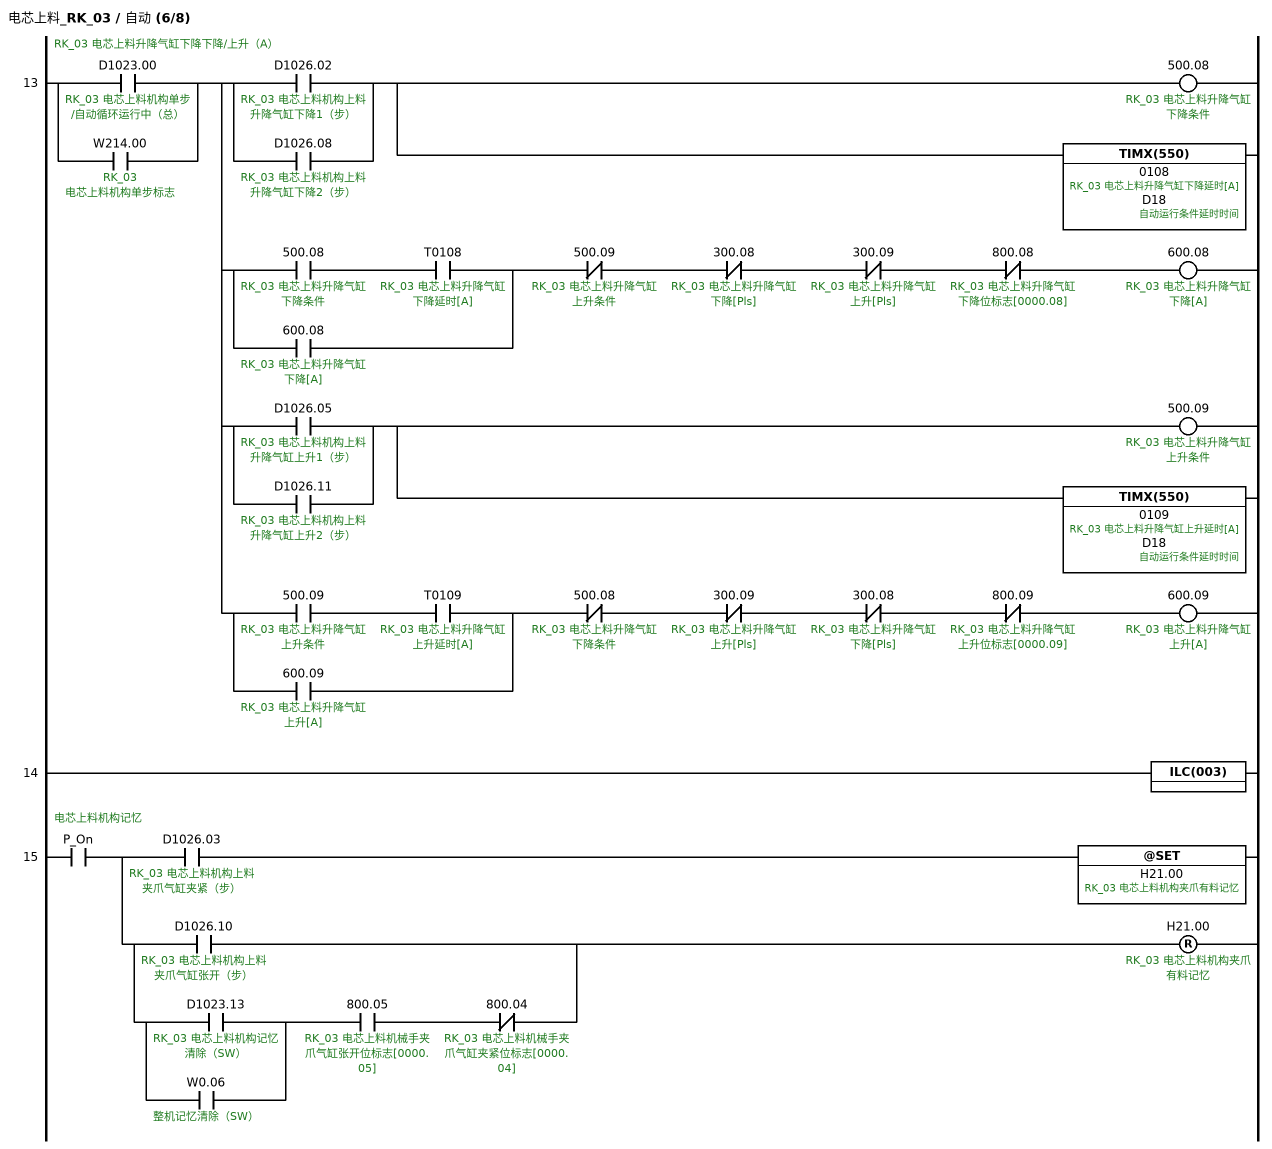
; [picture p384: 电芯上料_RK_03 / 自动, rungs 13-15]
; rung 13: RK_03 电芯上料升降气缸下降下降/上升（A）
LD D1023.00  ; RK_03 电芯上料机构单步/自动循环运行中（总）
OR W214.00  ; RK_03  电芯上料机构单步标志
OUT TR0
LD D1026.02  ; RK_03 电芯上料机构上料升降气缸下降1（步）
OR D1026.08  ; RK_03 电芯上料机构上料升降气缸下降2（步）
ANDLD
OUT 500.08  ; RK_03 电芯上料升降气缸下降条件
TIMX(550) 0108 D18  ; 自动运行条件延时时间, RK_03 电芯上料升降气缸下降延时[A]
LD TR0
LD 500.08  ; RK_03 电芯上料升降气缸下降条件
AND T0108  ; RK_03 电芯上料升降气缸下降延时[A]
OR 600.08  ; RK_03 电芯上料升降气缸下降[A]
ANDLD
ANDNOT 500.09  ; RK_03 电芯上料升降气缸上升条件
ANDNOT 300.08  ; RK_03 电芯上料升降气缸下降[Pls]
ANDNOT 300.09  ; RK_03 电芯上料升降气缸上升[Pls]
ANDNOT 800.08  ; RK_03 电芯上料升降气缸下降位标志[0000.08]
OUT 600.08  ; RK_03 电芯上料升降气缸下降[A]
LD TR0
LD D1026.05  ; RK_03 电芯上料机构上料升降气缸上升1（步）
OR D1026.11  ; RK_03 电芯上料机构上料升降气缸上升2（步）
ANDLD
OUT 500.09  ; RK_03 电芯上料升降气缸上升条件
TIMX(550) 0109 D18  ; 自动运行条件延时时间, RK_03 电芯上料升降气缸上升延时[A]
LD TR0
LD 500.09  ; RK_03 电芯上料升降气缸上升条件
AND T0109  ; RK_03 电芯上料升降气缸上升延时[A]
OR 600.09  ; RK_03 电芯上料升降气缸上升[A]
ANDLD
ANDNOT 500.08  ; RK_03 电芯上料升降气缸下降条件
ANDNOT 300.09  ; RK_03 电芯上料升降气缸上升[Pls]
ANDNOT 300.08  ; RK_03 电芯上料升降气缸下降[Pls]
ANDNOT 800.09  ; RK_03 电芯上料升降气缸上升位标志[0000.09]
OUT 600.09  ; RK_03 电芯上料升降气缸上升[A]
; rung 14
ILC(003)
; rung 15: 电芯上料机构记忆
LD P_On
OUT TR0
AND D1026.03  ; RK_03 电芯上料机构上料夹爪气缸夹紧（步）
@SET H21.00  ; RK_03 电芯上料机构夹爪有料记忆
LD TR0
LD D1026.10  ; RK_03 电芯上料机构上料夹爪气缸张开（步）
LD D1023.13  ; RK_03 电芯上料机构记忆清除（SW）
OR W0.06  ; 整机记忆清除（SW）
AND 800.05  ; RK_03 电芯上料机械手夹爪气缸张开位标志[0000.05]
ANDNOT 800.04  ; RK_03 电芯上料机械手夹爪气缸夹紧位标志[0000.04]
ORLD
ANDLD
RSET H21.00  ; RK_03 电芯上料机构夹爪有料记忆

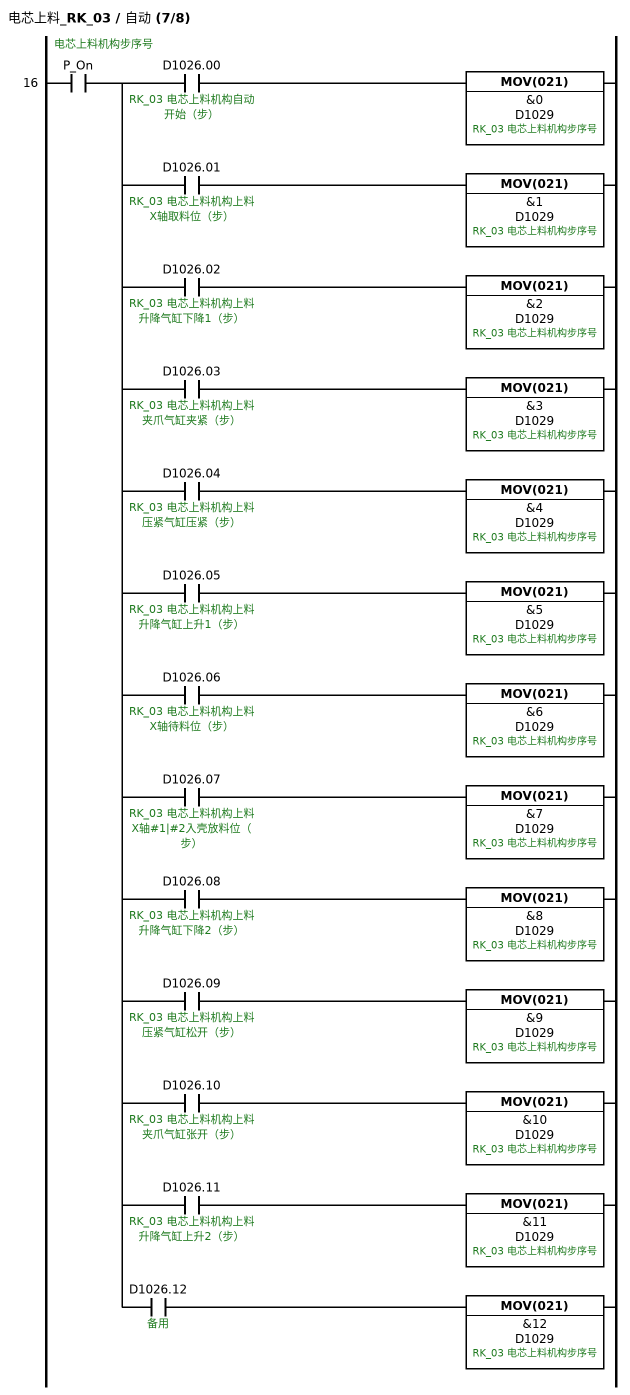
; rung 16: 电芯上料机构步序号
LD P_On
OUT TR0
AND D1026.00  ; RK_03 电芯上料机构自动开始（步）
MOV(021) &0 D1029  ; RK_03 电芯上料机构步序号
LD TR0
AND D1026.01  ; RK_03 电芯上料机构上料X轴取料位（步）
MOV(021) &1 D1029  ; RK_03 电芯上料机构步序号
LD TR0
AND D1026.02  ; RK_03 电芯上料机构上料升降气缸下降1（步）
MOV(021) &2 D1029  ; RK_03 电芯上料机构步序号
LD TR0
AND D1026.03  ; RK_03 电芯上料机构上料夹爪气缸夹紧（步）
MOV(021) &3 D1029  ; RK_03 电芯上料机构步序号
LD TR0
AND D1026.04  ; RK_03 电芯上料机构上料压紧气缸压紧（步）
MOV(021) &4 D1029  ; RK_03 电芯上料机构步序号
LD TR0
AND D1026.05  ; RK_03 电芯上料机构上料升降气缸上升1（步）
MOV(021) &5 D1029  ; RK_03 电芯上料机构步序号
LD TR0
AND D1026.06  ; RK_03 电芯上料机构上料X轴待料位（步）
MOV(021) &6 D1029  ; RK_03 电芯上料机构步序号
LD TR0
AND D1026.07  ; RK_03 电芯上料机构上料X轴#1|#2入壳放料位（步）
MOV(021) &7 D1029  ; RK_03 电芯上料机构步序号
LD TR0
AND D1026.08  ; RK_03 电芯上料机构上料升降气缸下降2（步）
MOV(021) &8 D1029  ; RK_03 电芯上料机构步序号
LD TR0
AND D1026.09  ; RK_03 电芯上料机构上料压紧气缸松开（步）
MOV(021) &9 D1029  ; RK_03 电芯上料机构步序号
LD TR0
AND D1026.10  ; RK_03 电芯上料机构上料夹爪气缸张开（步）
MOV(021) &10 D1029  ; RK_03 电芯上料机构步序号
LD TR0
AND D1026.11  ; RK_03 电芯上料机构上料升降气缸上升2（步）
MOV(021) &11 D1029  ; RK_03 电芯上料机构步序号
LD TR0
AND D1026.12  ; 备用
MOV(021) &12 D1029  ; RK_03 电芯上料机构步序号

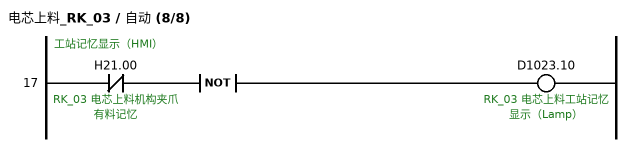
; rung 17: 工站记忆显示（HMI）
LDNOT H21.00  ; RK_03 电芯上料机构夹爪有料记忆
NOT(520)
OUT D1023.10  ; RK_03 电芯上料工站记忆显示（Lamp）

### Section 复位

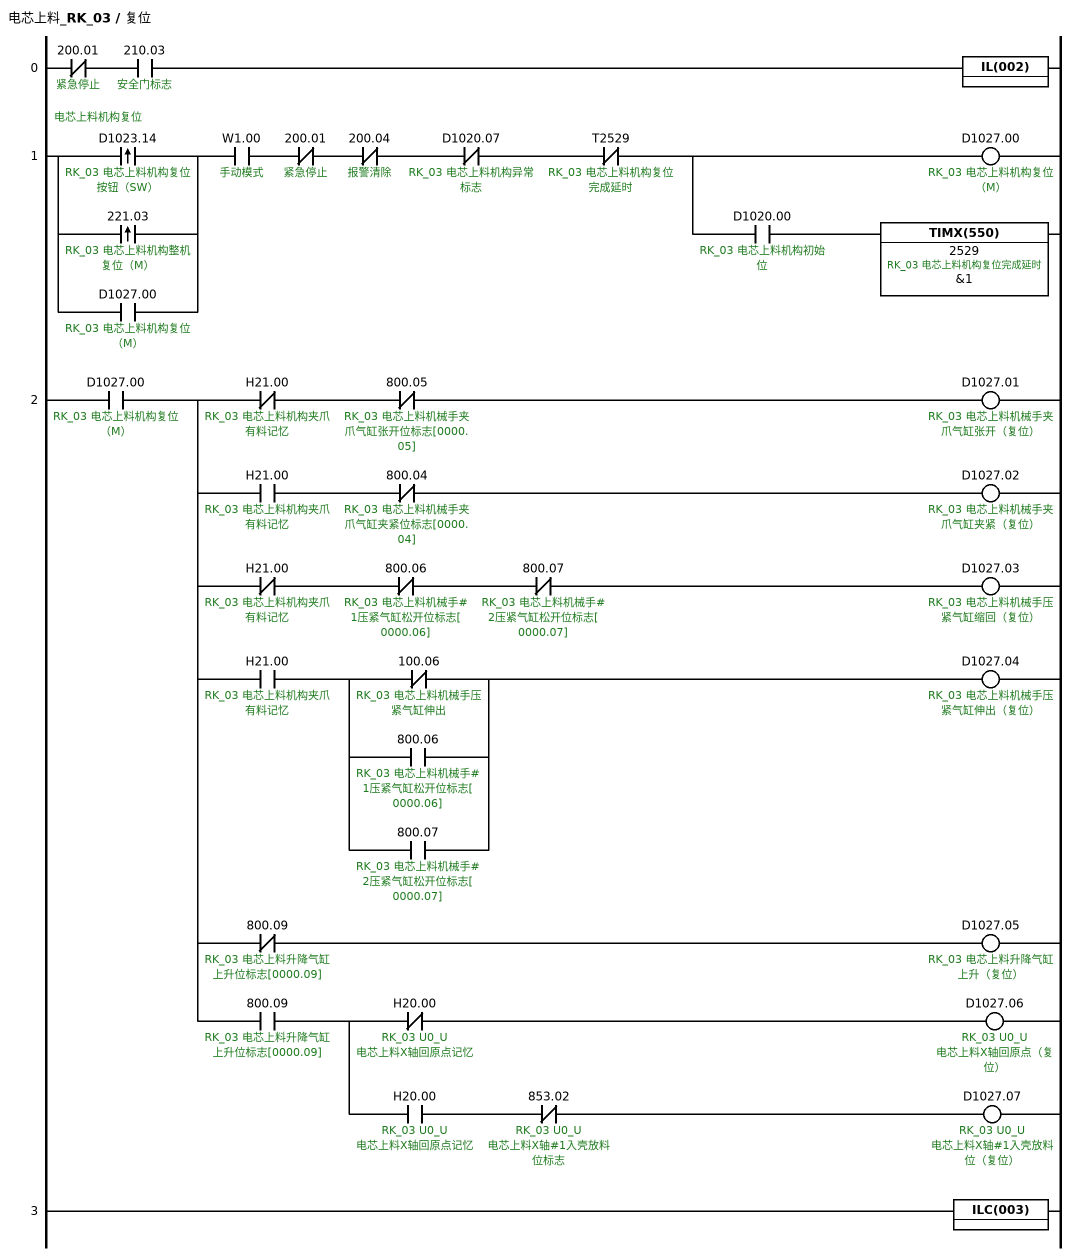
; rung 0
LDNOT 200.01  ; 紧急停止
AND 210.03  ; 安全门标志
IL(002)
; rung 1: 电芯上料机构复位
@LD D1023.14  ; RK_03 电芯上料机构复位按钮（SW）
@OR 221.03  ; RK_03 电芯上料机构整机复位（M）
OR D1027.00  ; RK_03 电芯上料机构复位（M）
AND W1.00  ; 手动模式
ANDNOT 200.01  ; 紧急停止
ANDNOT 200.04  ; 报警清除
ANDNOT D1020.07  ; RK_03 电芯上料机构异常标志
ANDNOT T2529  ; RK_03 电芯上料机构复位完成延时
OUT D1027.00  ; RK_03 电芯上料机构复位（M）
AND D1020.00  ; RK_03 电芯上料机构初始位
TIMX(550) 2529 &1  ; RK_03 电芯上料机构复位完成延时
; rung 2
LD D1027.00  ; RK_03 电芯上料机构复位（M）
OUT TR0
ANDNOT H21.00  ; RK_03 电芯上料机构夹爪有料记忆
ANDNOT 800.05  ; RK_03 电芯上料机械手夹爪气缸张开位标志[0000.05]
OUT D1027.01  ; RK_03 电芯上料机械手夹爪气缸张开（复位）
LD TR0
AND H21.00  ; RK_03 电芯上料机构夹爪有料记忆
ANDNOT 800.04  ; RK_03 电芯上料机械手夹爪气缸夹紧位标志[0000.04]
OUT D1027.02  ; RK_03 电芯上料机械手夹爪气缸夹紧（复位）
LD TR0
ANDNOT H21.00  ; RK_03 电芯上料机构夹爪有料记忆
ANDNOT 800.06  ; RK_03 电芯上料机械手#1压紧气缸松开位标志[0000.06]
ANDNOT 800.07  ; RK_03 电芯上料机械手#2压紧气缸松开位标志[0000.07]
OUT D1027.03  ; RK_03 电芯上料机械手压紧气缸缩回（复位）
LD TR0
AND H21.00  ; RK_03 电芯上料机构夹爪有料记忆
LDNOT 100.06  ; RK_03 电芯上料机械手压紧气缸伸出
OR 800.06  ; RK_03 电芯上料机械手#1压紧气缸松开位标志[0000.06]
OR 800.07  ; RK_03 电芯上料机械手#2压紧气缸松开位标志[0000.07]
ANDLD
OUT D1027.04  ; RK_03 电芯上料机械手压紧气缸伸出（复位）
LD TR0
ANDNOT 800.09  ; RK_03 电芯上料升降气缸上升位标志[0000.09]
OUT D1027.05  ; RK_03 电芯上料升降气缸上升（复位）
LD TR0
AND 800.09  ; RK_03 电芯上料升降气缸上升位标志[0000.09]
OUT TR0
ANDNOT H20.00  ; RK_03 U0_U 电芯上料X轴回原点记忆
OUT D1027.06  ; RK_03 U0_U 电芯上料X轴回原点（复位）
LD TR0
AND H20.00  ; RK_03 U0_U 电芯上料X轴回原点记忆
ANDNOT 853.02  ; RK_03 U0_U 电芯上料X轴#1入壳放料位标志
OUT D1027.07  ; RK_03 U0_U 电芯上料X轴#1入壳放料位（复位）
; rung 3
ILC(003)

### Section 指示灯

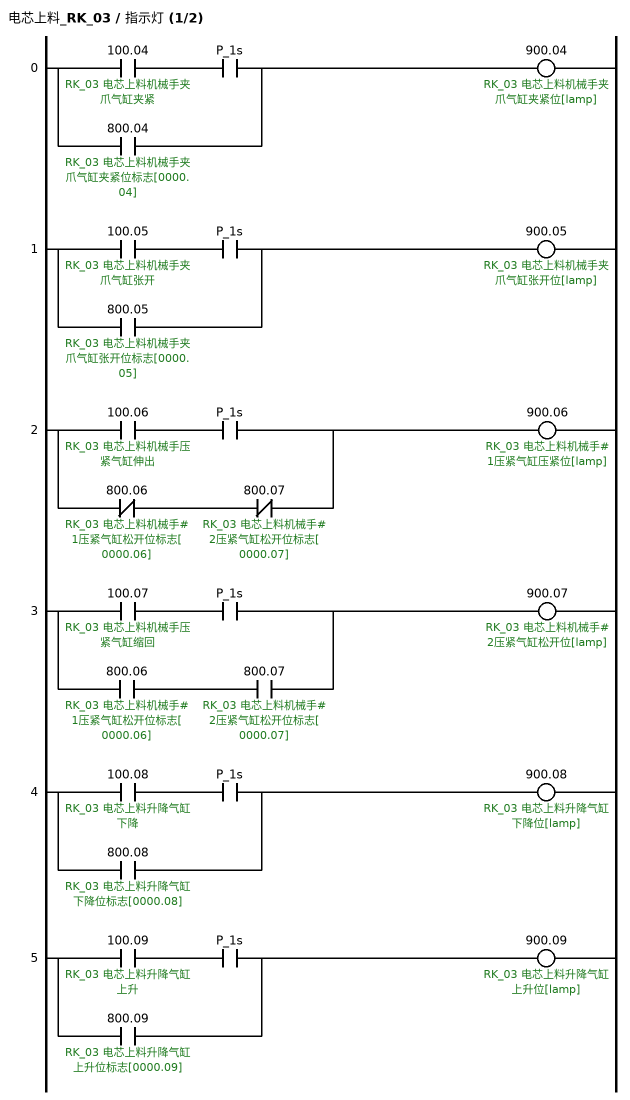
; rung 0
LD 100.04  ; RK_03 电芯上料机械手夹爪气缸夹紧
AND P_1s
OR 800.04  ; RK_03 电芯上料机械手夹爪气缸夹紧位标志[0000.04]
OUT 900.04  ; RK_03 电芯上料机械手夹爪气缸夹紧位[lamp]
; rung 1
LD 100.05  ; RK_03 电芯上料机械手夹爪气缸张开
AND P_1s
OR 800.05  ; RK_03 电芯上料机械手夹爪气缸张开位标志[0000.05]
OUT 900.05  ; RK_03 电芯上料机械手夹爪气缸张开位[lamp]
; rung 2
LD 100.06  ; RK_03 电芯上料机械手压紧气缸伸出
AND P_1s
LDNOT 800.06  ; RK_03 电芯上料机械手#1压紧气缸松开位标志[0000.06]
ANDNOT 800.07  ; RK_03 电芯上料机械手#2压紧气缸松开位标志[0000.07]
ORLD
OUT 900.06  ; RK_03 电芯上料机械手#1压紧气缸压紧位[lamp]
; rung 3
LD 100.07  ; RK_03 电芯上料机械手压紧气缸缩回
AND P_1s
LD 800.06  ; RK_03 电芯上料机械手#1压紧气缸松开位标志[0000.06]
AND 800.07  ; RK_03 电芯上料机械手#2压紧气缸松开位标志[0000.07]
ORLD
OUT 900.07  ; RK_03 电芯上料机械手#2压紧气缸松开位[lamp]
; rung 4
LD 100.08  ; RK_03 电芯上料升降气缸下降
AND P_1s
OR 800.08  ; RK_03 电芯上料升降气缸下降位标志[0000.08]
OUT 900.08  ; RK_03 电芯上料升降气缸下降位[lamp]
; rung 5
LD 100.09  ; RK_03 电芯上料升降气缸上升
AND P_1s
OR 800.09  ; RK_03 电芯上料升降气缸上升位标志[0000.09]
OUT 900.09  ; RK_03 电芯上料升降气缸上升位[lamp]

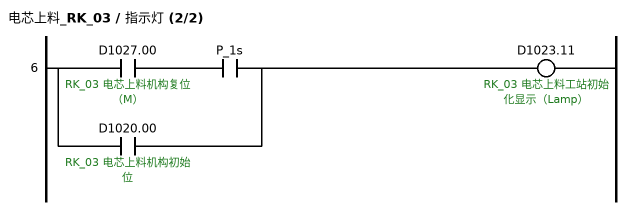
; rung 6
LD D1027.00  ; RK_03 电芯上料机构复位（M）
AND P_1s
OR D1020.00  ; RK_03 电芯上料机构初始位
OUT D1023.11  ; RK_03 电芯上料工站初始化显示（Lamp）

### Section 外部输出

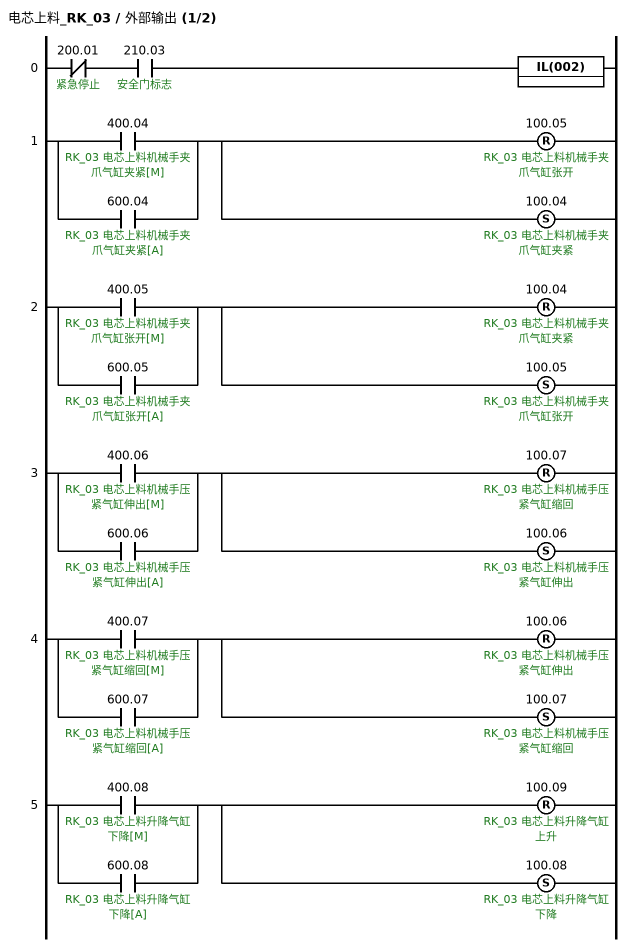
; rung 0
LDNOT 200.01  ; 紧急停止
AND 210.03  ; 安全门标志
IL(002)
; rung 1
LD 400.04  ; RK_03 电芯上料机械手夹爪气缸夹紧[M]
OR 600.04  ; RK_03 电芯上料机械手夹爪气缸夹紧[A]
RSET 100.05  ; RK_03 电芯上料机械手夹爪气缸张开
SET 100.04  ; RK_03 电芯上料机械手夹爪气缸夹紧
; rung 2
LD 400.05  ; RK_03 电芯上料机械手夹爪气缸张开[M]
OR 600.05  ; RK_03 电芯上料机械手夹爪气缸张开[A]
RSET 100.04  ; RK_03 电芯上料机械手夹爪气缸夹紧
SET 100.05  ; RK_03 电芯上料机械手夹爪气缸张开
; rung 3
LD 400.06  ; RK_03 电芯上料机械手压紧气缸伸出[M]
OR 600.06  ; RK_03 电芯上料机械手压紧气缸伸出[A]
RSET 100.07  ; RK_03 电芯上料机械手压紧气缸缩回
SET 100.06  ; RK_03 电芯上料机械手压紧气缸伸出
; rung 4
LD 400.07  ; RK_03 电芯上料机械手压紧气缸缩回[M]
OR 600.07  ; RK_03 电芯上料机械手压紧气缸缩回[A]
RSET 100.06  ; RK_03 电芯上料机械手压紧气缸伸出
SET 100.07  ; RK_03 电芯上料机械手压紧气缸缩回
; rung 5
LD 400.08  ; RK_03 电芯上料升降气缸下降[M]
OR 600.08  ; RK_03 电芯上料升降气缸下降[A]
RSET 100.09  ; RK_03 电芯上料升降气缸上升
SET 100.08  ; RK_03 电芯上料升降气缸下降

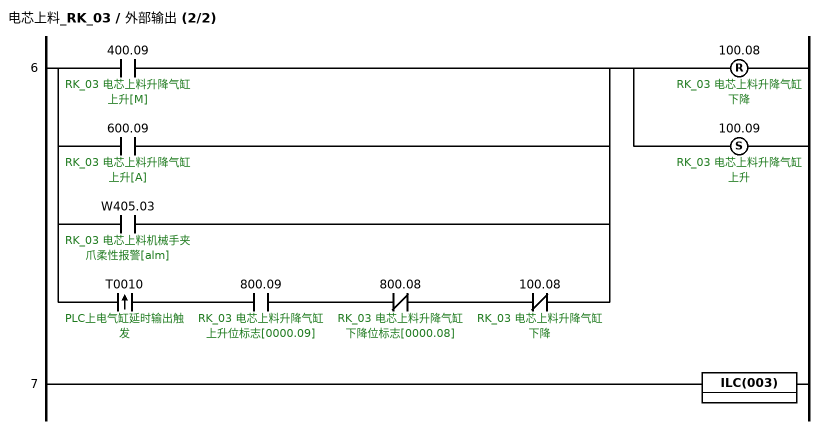
; rung 6
LD 400.09  ; RK_03 电芯上料升降气缸上升[M]
OR 600.09  ; RK_03 电芯上料升降气缸上升[A]
OR W405.03  ; RK_03 电芯上料机械手夹爪柔性报警[alm]
@LD T0010  ; PLC上电气缸延时输出触发
AND 800.09  ; RK_03 电芯上料升降气缸上升位标志[0000.09]
ANDNOT 800.08  ; RK_03 电芯上料升降气缸下降位标志[0000.08]
ANDNOT 100.08  ; RK_03 电芯上料升降气缸下降
ORLD
RSET 100.08  ; RK_03 电芯上料升降气缸下降
SET 100.09  ; RK_03 电芯上料升降气缸上升
; rung 7
ILC(003)

### Section END
; rung 0
END(001)

## Program 电芯除尘_RK_04 (cyclic task 4)

### Section Main

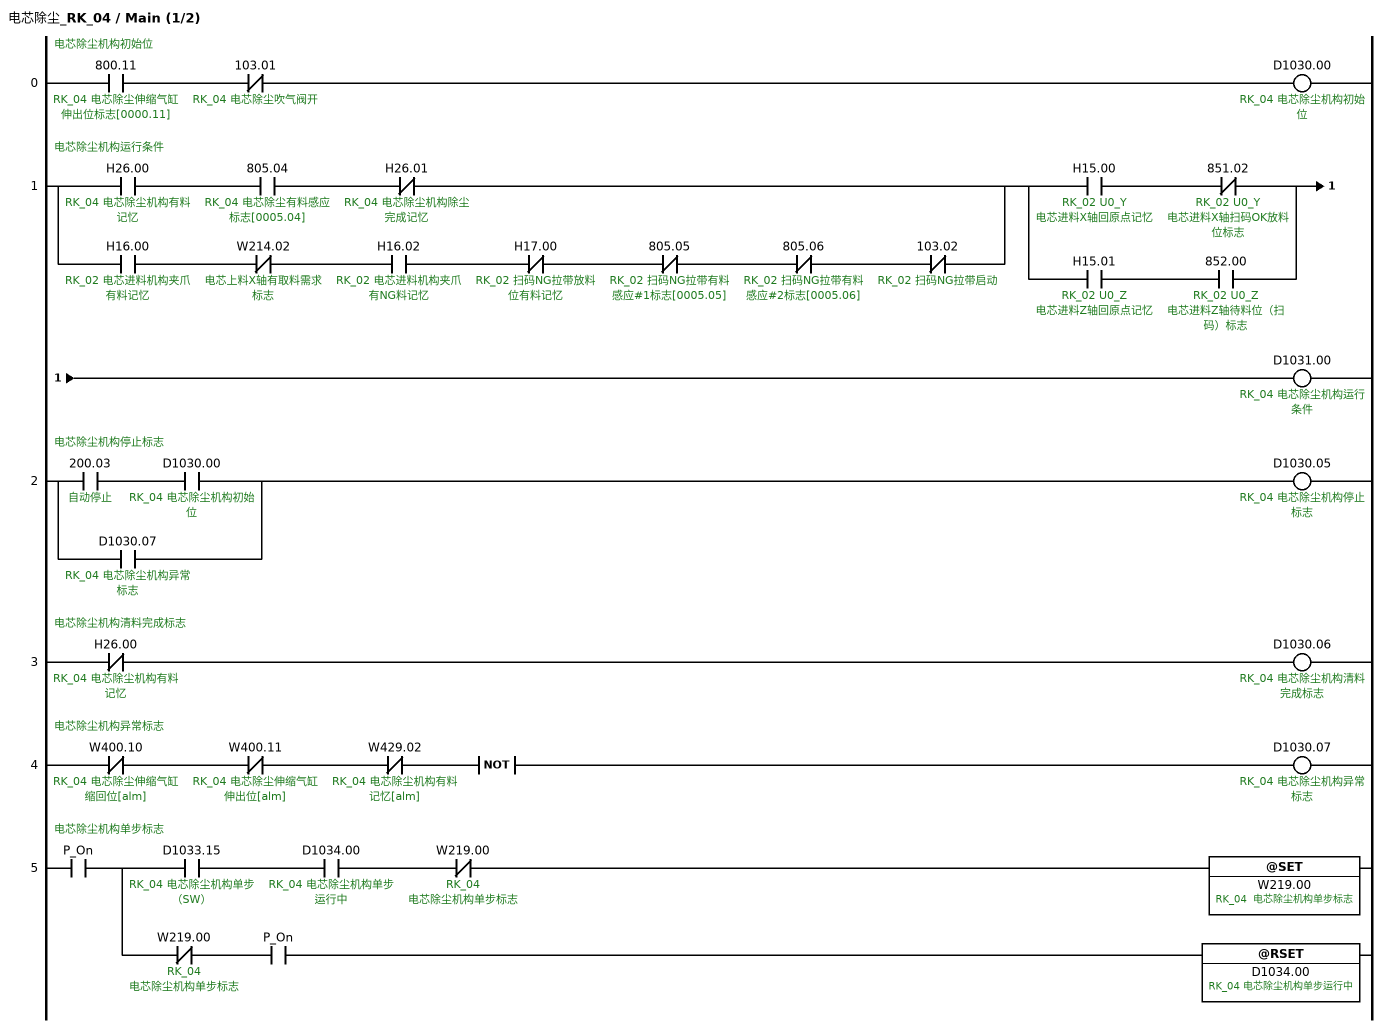
; rung 0: 电芯除尘机构初始位
LD 800.11  ; RK_04 电芯除尘伸缩气缸伸出位标志[0000.11]
ANDNOT 103.01  ; RK_04 电芯除尘吹气阀开
OUT D1030.00  ; RK_04 电芯除尘机构初始位
; rung 1: 电芯除尘机构运行条件
LD H26.00  ; RK_04 电芯除尘机构有料记忆  // 正常上料完成工况！
AND 805.04  ; RK_04 电芯除尘有料感应标志[0005.04]
ANDNOT H26.01  ; RK_04 电芯除尘机构除尘完成记忆
LD H16.00  ; RK_02 电芯进料机构夹爪有料记忆  // 电芯进料X轴有NG料&NG拉带允许上料&电芯上料X轴没有上料需求，则电芯进料X轴下NG料，此时电芯除尘机构动作！！
ANDNOT W214.02  ; 电芯上料X轴有取料需求标志
AND H16.02  ; RK_02 电芯进料机构夹爪有NG料记忆
ANDNOT H17.00  ; RK_02 扫码NG拉带放料位有料记忆
ANDNOT 805.05  ; RK_02 扫码NG拉带有料感应#1标志[0005.05]
ANDNOT 805.06  ; RK_02 扫码NG拉带有料感应#2标志[0005.06]
ANDNOT 103.02  ; RK_02 扫码NG拉带启动
ORLD
LD H15.00  ; RK_02 U0_Y 电芯进料X轴回原点记忆
ANDNOT 851.02  ; RK_02 U0_Y 电芯进料X轴扫码OK放料位标志
LD H15.01  ; RK_02 U0_Z 电芯进料Z轴回原点记忆
AND 852.00  ; RK_02 U0_Z 电芯进料Z轴待料位（扫码）标志
ORLD
ANDLD
OUT D1031.00  ; RK_04 电芯除尘机构运行条件
; rung 2: 电芯除尘机构停止标志
LD 200.03  ; 自动停止
AND D1030.00  ; RK_04 电芯除尘机构初始位
OR D1030.07  ; RK_04 电芯除尘机构异常标志
OUT D1030.05  ; RK_04 电芯除尘机构停止标志
; rung 3: 电芯除尘机构清料完成标志
LDNOT H26.00  ; RK_04 电芯除尘机构有料记忆
OUT D1030.06  ; RK_04 电芯除尘机构清料完成标志
; rung 4: 电芯除尘机构异常标志
LDNOT W400.10  ; RK_04 电芯除尘伸缩气缸缩回位[alm]
ANDNOT W400.11  ; RK_04 电芯除尘伸缩气缸伸出位[alm]
ANDNOT W429.02  ; RK_04 电芯除尘机构有料记忆[alm]
NOT(520)
OUT D1030.07  ; RK_04 电芯除尘机构异常标志
; rung 5: 电芯除尘机构单步标志
LD P_On
OUT TR0
AND D1033.15  ; RK_04 电芯除尘机构单步（SW）
AND D1034.00  ; RK_04 电芯除尘机构单步运行中
ANDNOT W219.00  ; RK_04  电芯除尘机构单步标志
@SET W219.00  ; RK_04  电芯除尘机构单步标志
LD TR0
ANDNOT W219.00  ; RK_04  电芯除尘机构单步标志
AND P_On
@RSET D1034.00  ; RK_04 电芯除尘机构单步运行中

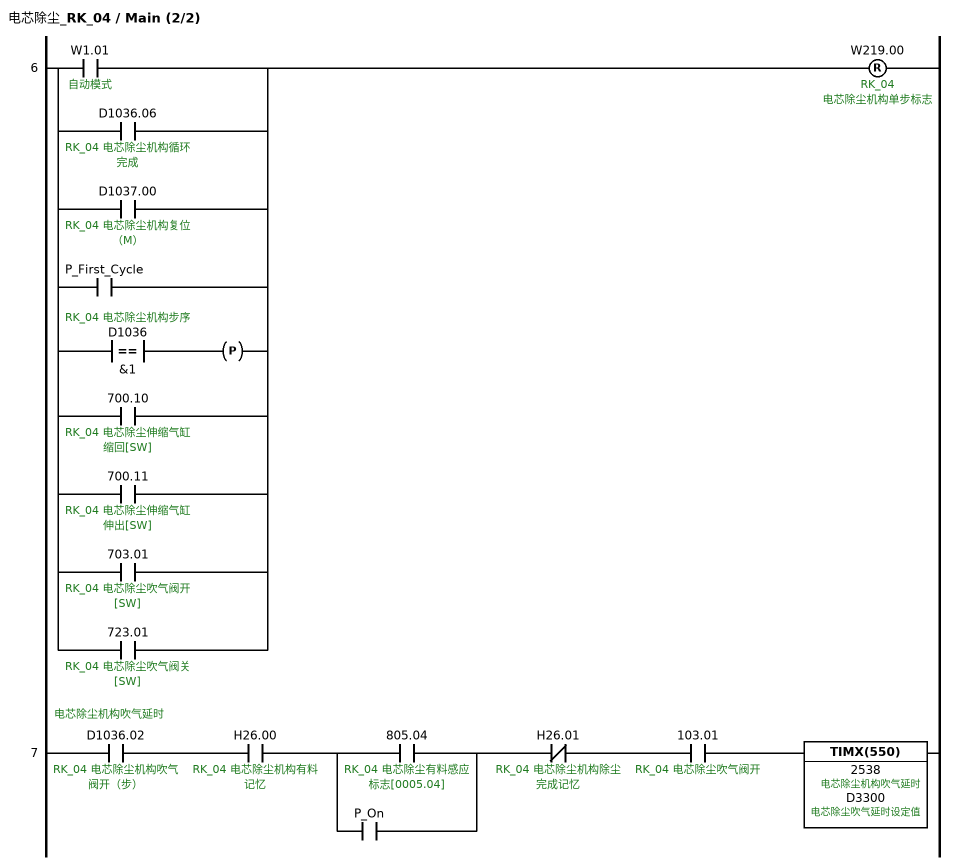
; rung 6
LD W1.01  ; 自动模式
OR D1036.06  ; RK_04 电芯除尘机构循环完成
OR D1037.00  ; RK_04 电芯除尘机构复位（M）
OR P_First_Cycle
LD=(300) D1036 &1  ; RK_04 电芯除尘机构步序
UP(521)
ORLD
OR 700.10  ; RK_04 电芯除尘伸缩气缸缩回[SW]
OR 700.11  ; RK_04 电芯除尘伸缩气缸伸出[SW]
OR 703.01  ; RK_04 电芯除尘吹气阀开[SW]
OR 723.01  ; RK_04 电芯除尘吹气阀关[SW]
RSET W219.00  ; RK_04  电芯除尘机构单步标志
; rung 7: 电芯除尘机构吹气延时
LD D1036.02  ; RK_04 电芯除尘机构吹气阀开（步）
AND H26.00  ; RK_04 电芯除尘机构有料记忆
LD 805.04  ; RK_04 电芯除尘有料感应标志[0005.04]
OR P_On
ANDLD
ANDNOT H26.01  ; RK_04 电芯除尘机构除尘完成记忆
AND 103.01  ; RK_04 电芯除尘吹气阀开
TIMX(550) 2538 D3300  ; 电芯除尘吹气延时设定值, 电芯除尘机构吹气延时

### Section 手动

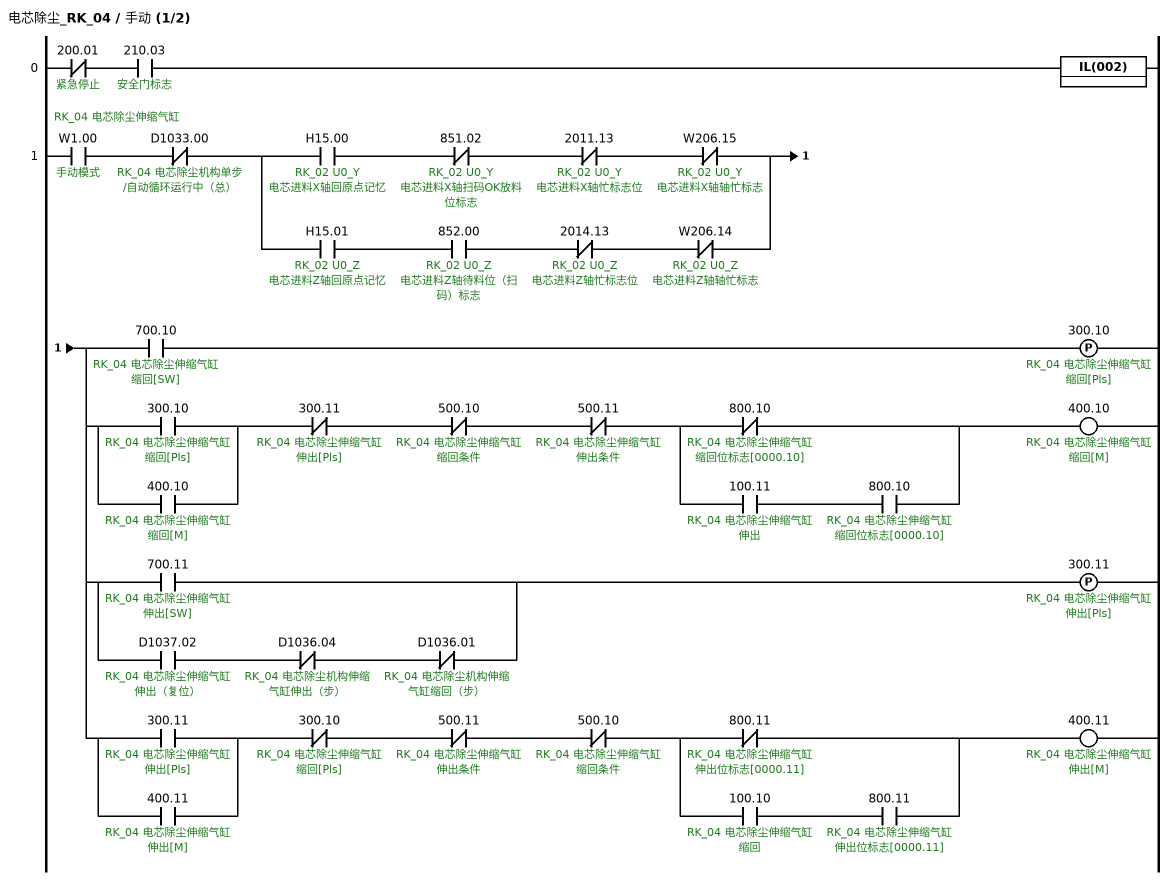
; rung 0
LDNOT 200.01  ; 紧急停止
AND 210.03  ; 安全门标志
IL(002)
; rung 1: RK_04 电芯除尘伸缩气缸
LD W1.00  ; 手动模式
ANDNOT D1033.00  ; RK_04 电芯除尘机构单步/自动循环运行中（总）
LD H15.00  ; RK_02 U0_Y 电芯进料X轴回原点记忆
ANDNOT 851.02  ; RK_02 U0_Y 电芯进料X轴扫码OK放料位标志
ANDNOT 2011.13  ; RK_02 U0_Y 电芯进料X轴忙标志位
ANDNOT W206.15  ; RK_02 U0_Y 电芯进料X轴轴忙标志
LD H15.01  ; RK_02 U0_Z 电芯进料Z轴回原点记忆
AND 852.00  ; RK_02 U0_Z 电芯进料Z轴待料位（扫码）标志
ANDNOT 2014.13  ; RK_02 U0_Z 电芯进料Z轴忙标志位
ANDNOT W206.14  ; RK_02 U0_Z 电芯进料Z轴轴忙标志
ORLD
ANDLD
OUT TR0
AND 700.10  ; RK_04 电芯除尘伸缩气缸缩回[SW]
DIFU(013) 300.10  ; RK_04 电芯除尘伸缩气缸缩回[Pls]
LD TR0
LD 300.10  ; RK_04 电芯除尘伸缩气缸缩回[Pls]
OR 400.10  ; RK_04 电芯除尘伸缩气缸缩回[M]
ANDLD
ANDNOT 300.11  ; RK_04 电芯除尘伸缩气缸伸出[Pls]
ANDNOT 500.10  ; RK_04 电芯除尘伸缩气缸缩回条件
ANDNOT 500.11  ; RK_04 电芯除尘伸缩气缸伸出条件
LDNOT 800.10  ; RK_04 电芯除尘伸缩气缸缩回位标志[0000.10]
LD 100.11  ; RK_04 电芯除尘伸缩气缸伸出
AND 800.10  ; RK_04 电芯除尘伸缩气缸缩回位标志[0000.10]
ORLD
ANDLD
OUT 400.10  ; RK_04 电芯除尘伸缩气缸缩回[M]
LD TR0
LD 700.11  ; RK_04 电芯除尘伸缩气缸伸出[SW]
LD D1037.02  ; RK_04 电芯除尘伸缩气缸伸出（复位）
ANDNOT D1036.04  ; RK_04 电芯除尘机构伸缩气缸伸出（步）
ANDNOT D1036.01  ; RK_04 电芯除尘机构伸缩气缸缩回（步）
ORLD
ANDLD
DIFU(013) 300.11  ; RK_04 电芯除尘伸缩气缸伸出[Pls]
LD TR0
LD 300.11  ; RK_04 电芯除尘伸缩气缸伸出[Pls]
OR 400.11  ; RK_04 电芯除尘伸缩气缸伸出[M]
ANDLD
ANDNOT 300.10  ; RK_04 电芯除尘伸缩气缸缩回[Pls]
ANDNOT 500.11  ; RK_04 电芯除尘伸缩气缸伸出条件
ANDNOT 500.10  ; RK_04 电芯除尘伸缩气缸缩回条件
LDNOT 800.11  ; RK_04 电芯除尘伸缩气缸伸出位标志[0000.11]
LD 100.10  ; RK_04 电芯除尘伸缩气缸缩回
AND 800.11  ; RK_04 电芯除尘伸缩气缸伸出位标志[0000.11]
ORLD
ANDLD
OUT 400.11  ; RK_04 电芯除尘伸缩气缸伸出[M]

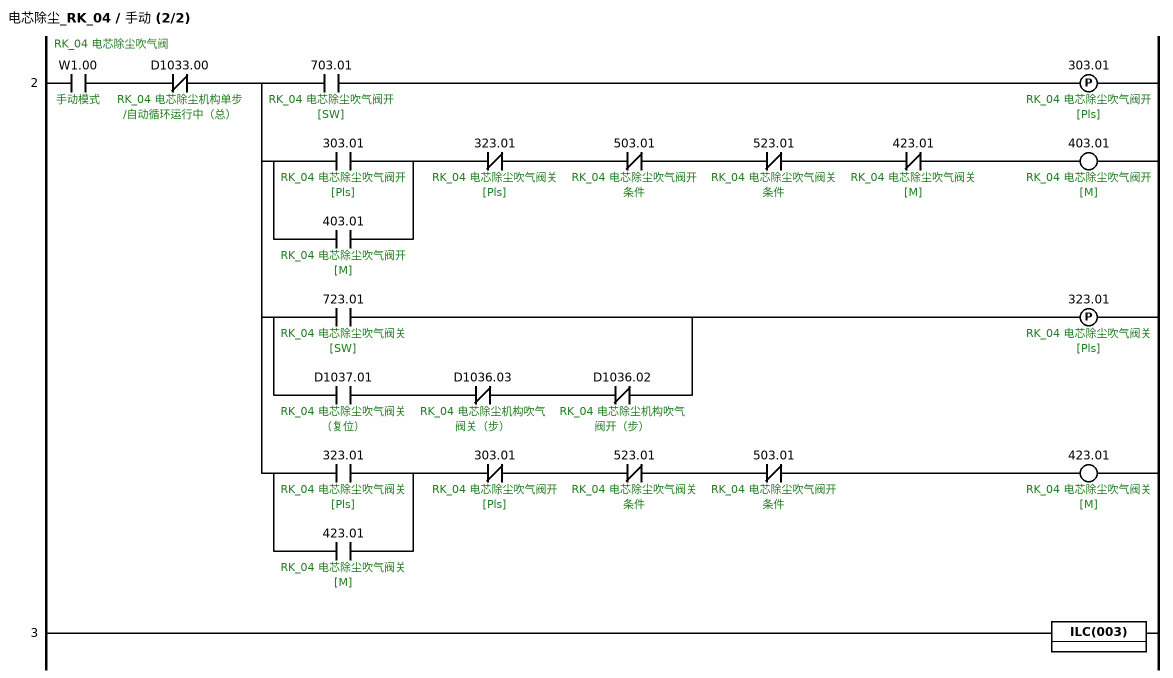
; rung 2: RK_04 电芯除尘吹气阀
LD W1.00  ; 手动模式
ANDNOT D1033.00  ; RK_04 电芯除尘机构单步/自动循环运行中（总）
OUT TR0
AND 703.01  ; RK_04 电芯除尘吹气阀开[SW]
DIFU(013) 303.01  ; RK_04 电芯除尘吹气阀开[Pls]
LD TR0
LD 303.01  ; RK_04 电芯除尘吹气阀开[Pls]
OR 403.01  ; RK_04 电芯除尘吹气阀开[M]
ANDLD
ANDNOT 323.01  ; RK_04 电芯除尘吹气阀关[Pls]
ANDNOT 503.01  ; RK_04 电芯除尘吹气阀开条件
ANDNOT 523.01  ; RK_04 电芯除尘吹气阀关条件
ANDNOT 423.01  ; RK_04 电芯除尘吹气阀关[M]
OUT 403.01  ; RK_04 电芯除尘吹气阀开[M]
LD TR0
LD 723.01  ; RK_04 电芯除尘吹气阀关[SW]
LD D1037.01  ; RK_04 电芯除尘吹气阀关（复位）
ANDNOT D1036.03  ; RK_04 电芯除尘机构吹气阀关（步）
ANDNOT D1036.02  ; RK_04 电芯除尘机构吹气阀开（步）
ORLD
ANDLD
DIFU(013) 323.01  ; RK_04 电芯除尘吹气阀关[Pls]
LD TR0
LD 323.01  ; RK_04 电芯除尘吹气阀关[Pls]
OR 423.01  ; RK_04 电芯除尘吹气阀关[M]
ANDLD
ANDNOT 303.01  ; RK_04 电芯除尘吹气阀开[Pls]
ANDNOT 523.01  ; RK_04 电芯除尘吹气阀关条件
ANDNOT 503.01  ; RK_04 电芯除尘吹气阀开条件
OUT 423.01  ; RK_04 电芯除尘吹气阀关[M]
; rung 3
ILC(003)

### Section 自动

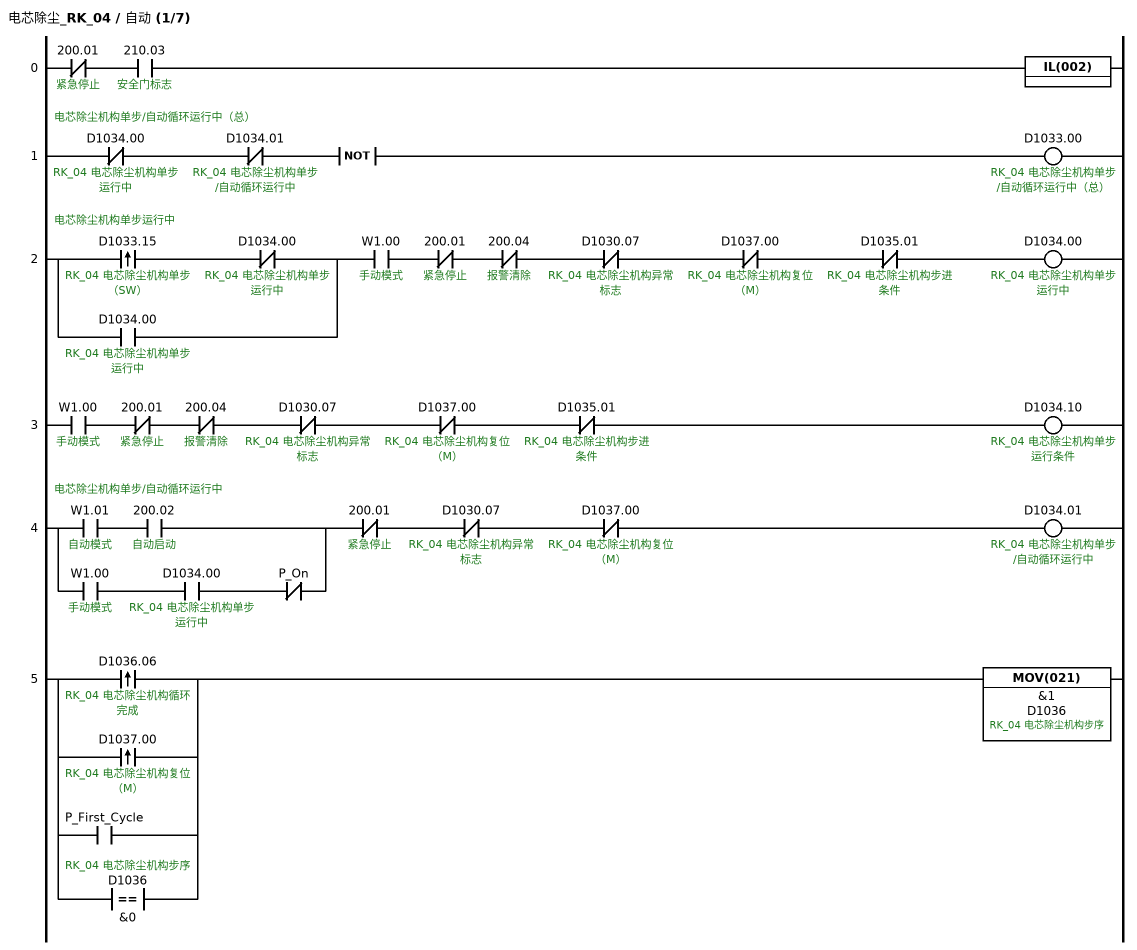
; rung 0
LDNOT 200.01  ; 紧急停止
AND 210.03  ; 安全门标志
IL(002)
; rung 1: 电芯除尘机构单步/自动循环运行中（总）
LDNOT D1034.00  ; RK_04 电芯除尘机构单步运行中
ANDNOT D1034.01  ; RK_04 电芯除尘机构单步/自动循环运行中
NOT(520)
OUT D1033.00  ; RK_04 电芯除尘机构单步/自动循环运行中（总）
; rung 2: 电芯除尘机构单步运行中
@LD D1033.15  ; RK_04 电芯除尘机构单步（SW）
ANDNOT D1034.00  ; RK_04 电芯除尘机构单步运行中
OR D1034.00  ; RK_04 电芯除尘机构单步运行中
AND W1.00  ; 手动模式
ANDNOT 200.01  ; 紧急停止
ANDNOT 200.04  ; 报警清除
ANDNOT D1030.07  ; RK_04 电芯除尘机构异常标志
ANDNOT D1037.00  ; RK_04 电芯除尘机构复位（M）
ANDNOT D1035.01  ; RK_04 电芯除尘机构步进条件
OUT D1034.00  ; RK_04 电芯除尘机构单步运行中
; rung 3
LD W1.00  ; 手动模式
ANDNOT 200.01  ; 紧急停止
ANDNOT 200.04  ; 报警清除
ANDNOT D1030.07  ; RK_04 电芯除尘机构异常标志
ANDNOT D1037.00  ; RK_04 电芯除尘机构复位（M）
ANDNOT D1035.01  ; RK_04 电芯除尘机构步进条件
OUT D1034.10  ; RK_04 电芯除尘机构单步运行条件
; rung 4: 电芯除尘机构单步/自动循环运行中
LD W1.01  ; 自动模式
AND 200.02  ; 自动启动
LD W1.00  ; 手动模式
AND D1034.00  ; RK_04 电芯除尘机构单步运行中
ANDNOT P_On
ORLD
ANDNOT 200.01  ; 紧急停止
ANDNOT D1030.07  ; RK_04 电芯除尘机构异常标志
ANDNOT D1037.00  ; RK_04 电芯除尘机构复位（M）
OUT D1034.01  ; RK_04 电芯除尘机构单步/自动循环运行中
; rung 5
@LD D1036.06  ; RK_04 电芯除尘机构循环完成
@OR D1037.00  ; RK_04 电芯除尘机构复位（M）
OR P_First_Cycle
OR=(300) D1036 &0  ; RK_04 电芯除尘机构步序
MOV(021) &1 D1036  ; RK_04 电芯除尘机构步序

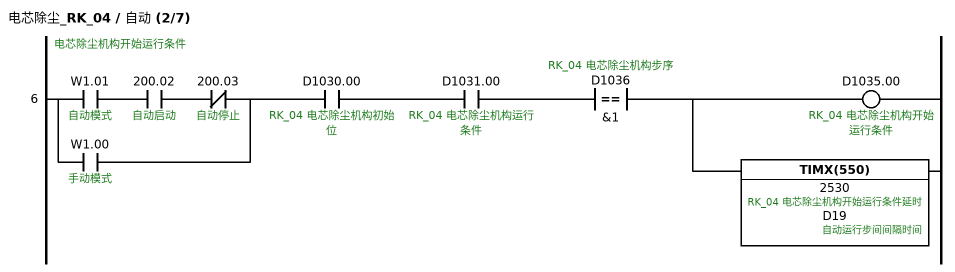
; rung 6: 电芯除尘机构开始运行条件
LD W1.01  ; 自动模式
AND 200.02  ; 自动启动
ANDNOT 200.03  ; 自动停止
OR W1.00  ; 手动模式
AND D1030.00  ; RK_04 电芯除尘机构初始位
AND D1031.00  ; RK_04 电芯除尘机构运行条件
AND=(300) D1036 &1  ; RK_04 电芯除尘机构步序
OUT D1035.00  ; RK_04 电芯除尘机构开始运行条件
TIMX(550) 2530 D19  ; 自动运行步间间隔时间, RK_04 电芯除尘机构开始运行条件延时

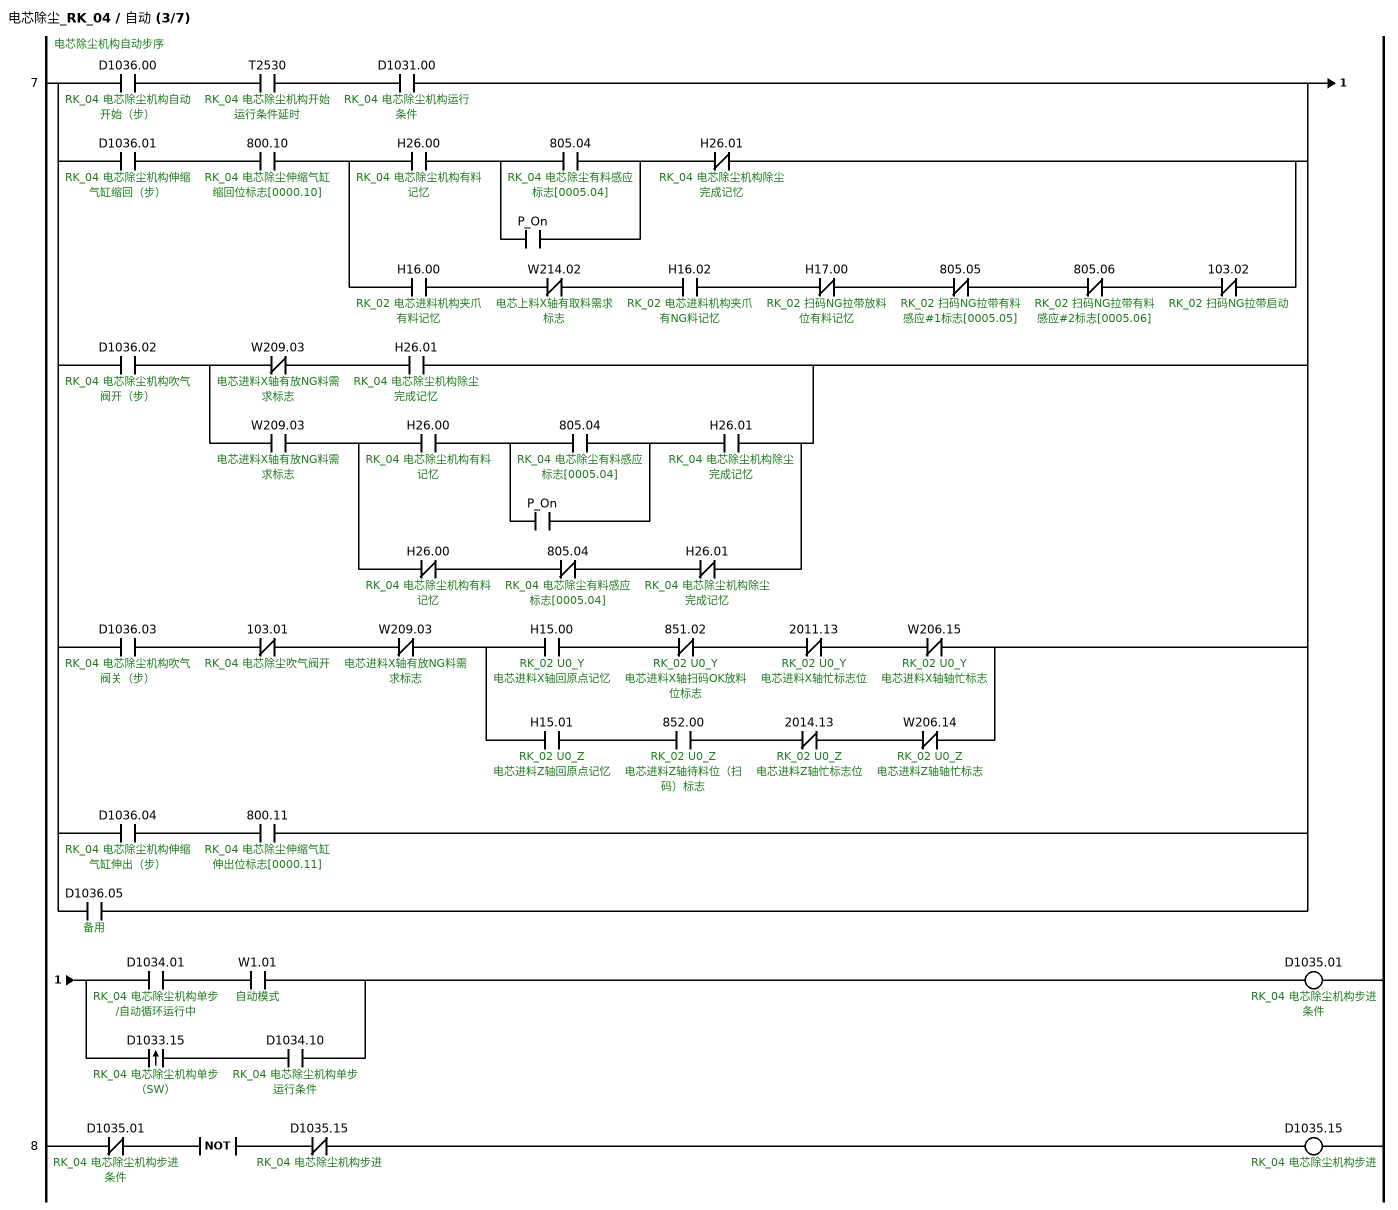
; rung 7: 电芯除尘机构自动步序
LD D1036.00  ; RK_04 电芯除尘机构自动开始（步）
AND T2530  ; RK_04 电芯除尘机构开始运行条件延时
AND D1031.00  ; RK_04 电芯除尘机构运行条件
LD D1036.01  ; RK_04 电芯除尘机构伸缩气缸缩回（步）
AND 800.10  ; RK_04 电芯除尘伸缩气缸缩回位标志[0000.10]
LD H26.00  ; RK_04 电芯除尘机构有料记忆  // 正常上料完成工况！
LD 805.04  ; RK_04 电芯除尘有料感应标志[0005.04]
OR P_On
ANDLD
ANDNOT H26.01  ; RK_04 电芯除尘机构除尘完成记忆
LD H16.00  ; RK_02 电芯进料机构夹爪有料记忆  // 电芯进料X轴有NG料&NG拉带允许上料&电芯上料X轴没有上料需求，则电芯进料X轴下NG料，此时电芯除尘机构动作！！
ANDNOT W214.02  ; 电芯上料X轴有取料需求标志
AND H16.02  ; RK_02 电芯进料机构夹爪有NG料记忆
ANDNOT H17.00  ; RK_02 扫码NG拉带放料位有料记忆
ANDNOT 805.05  ; RK_02 扫码NG拉带有料感应#1标志[0005.05]
ANDNOT 805.06  ; RK_02 扫码NG拉带有料感应#2标志[0005.06]
ANDNOT 103.02  ; RK_02 扫码NG拉带启动
ORLD
ANDLD
ORLD
LD D1036.02  ; RK_04 电芯除尘机构吹气阀开（步）
LDNOT W209.03  ; 电芯进料X轴有放NG料需求标志
AND H26.01  ; RK_04 电芯除尘机构除尘完成记忆
LD W209.03  ; 电芯进料X轴有放NG料需求标志
LD H26.00  ; RK_04 电芯除尘机构有料记忆
LD 805.04  ; RK_04 电芯除尘有料感应标志[0005.04]
OR P_On
ANDLD
AND H26.01  ; RK_04 电芯除尘机构除尘完成记忆
LDNOT H26.00  ; RK_04 电芯除尘机构有料记忆
ANDNOT 805.04  ; RK_04 电芯除尘有料感应标志[0005.04]
ANDNOT H26.01  ; RK_04 电芯除尘机构除尘完成记忆
ORLD
ANDLD
ORLD
ANDLD
ORLD
LD D1036.03  ; RK_04 电芯除尘机构吹气阀关（步）
ANDNOT 103.01  ; RK_04 电芯除尘吹气阀开
ANDNOT W209.03  ; 电芯进料X轴有放NG料需求标志
LD H15.00  ; RK_02 U0_Y 电芯进料X轴回原点记忆
ANDNOT 851.02  ; RK_02 U0_Y 电芯进料X轴扫码OK放料位标志
ANDNOT 2011.13  ; RK_02 U0_Y 电芯进料X轴忙标志位
ANDNOT W206.15  ; RK_02 U0_Y 电芯进料X轴轴忙标志
LD H15.01  ; RK_02 U0_Z 电芯进料Z轴回原点记忆
AND 852.00  ; RK_02 U0_Z 电芯进料Z轴待料位（扫码）标志
ANDNOT 2014.13  ; RK_02 U0_Z 电芯进料Z轴忙标志位
ANDNOT W206.14  ; RK_02 U0_Z 电芯进料Z轴轴忙标志
ORLD
ANDLD
ORLD
LD D1036.04  ; RK_04 电芯除尘机构伸缩气缸伸出（步）
AND 800.11  ; RK_04 电芯除尘伸缩气缸伸出位标志[0000.11]
ORLD
OR D1036.05  ; 备用
LD D1034.01  ; RK_04 电芯除尘机构单步/自动循环运行中
AND W1.01  ; 自动模式
@LD D1033.15  ; RK_04 电芯除尘机构单步（SW）
AND D1034.10  ; RK_04 电芯除尘机构单步运行条件
ORLD
ANDLD
OUT D1035.01  ; RK_04 电芯除尘机构步进条件
; rung 8
LDNOT D1035.01  ; RK_04 电芯除尘机构步进条件
NOT(520)
ANDNOT D1035.15  ; RK_04 电芯除尘机构步进
OUT D1035.15  ; RK_04 电芯除尘机构步进

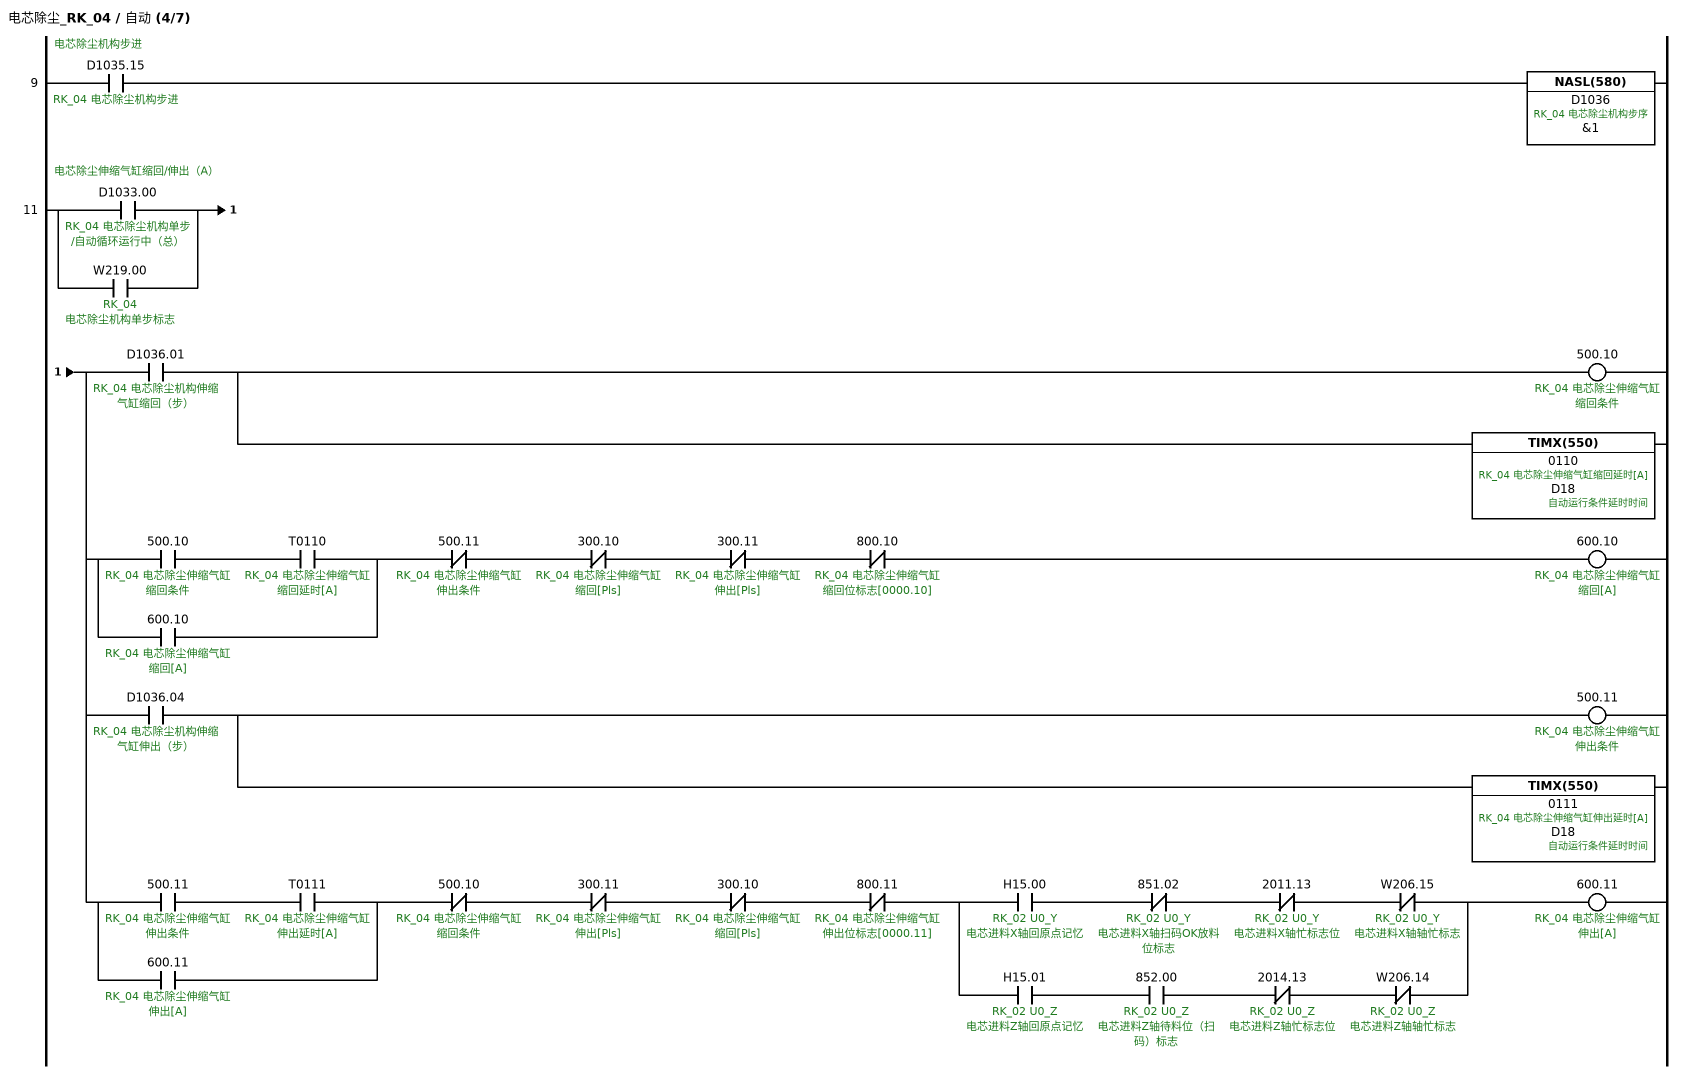
; rung 9: 电芯除尘机构步进
LD D1035.15  ; RK_04 电芯除尘机构步进
NASL(580) D1036 &1  ; RK_04 电芯除尘机构步序
; rung 10: 电芯除尘机构步序跳转
; rung 11: 电芯除尘伸缩气缸缩回/伸出（A）
LD D1033.00  ; RK_04 电芯除尘机构单步/自动循环运行中（总）
OR W219.00  ; RK_04  电芯除尘机构单步标志
OUT TR0
AND D1036.01  ; RK_04 电芯除尘机构伸缩气缸缩回（步）
OUT 500.10  ; RK_04 电芯除尘伸缩气缸缩回条件
TIMX(550) 0110 D18  ; 自动运行条件延时时间, RK_04 电芯除尘伸缩气缸缩回延时[A]
LD TR0
LD 500.10  ; RK_04 电芯除尘伸缩气缸缩回条件
AND T0110  ; RK_04 电芯除尘伸缩气缸缩回延时[A]
OR 600.10  ; RK_04 电芯除尘伸缩气缸缩回[A]
ANDLD
ANDNOT 500.11  ; RK_04 电芯除尘伸缩气缸伸出条件
ANDNOT 300.10  ; RK_04 电芯除尘伸缩气缸缩回[Pls]
ANDNOT 300.11  ; RK_04 电芯除尘伸缩气缸伸出[Pls]
ANDNOT 800.10  ; RK_04 电芯除尘伸缩气缸缩回位标志[0000.10]
OUT 600.10  ; RK_04 电芯除尘伸缩气缸缩回[A]
LD TR0
AND D1036.04  ; RK_04 电芯除尘机构伸缩气缸伸出（步）
OUT 500.11  ; RK_04 电芯除尘伸缩气缸伸出条件
TIMX(550) 0111 D18  ; 自动运行条件延时时间, RK_04 电芯除尘伸缩气缸伸出延时[A]
LD TR0
LD 500.11  ; RK_04 电芯除尘伸缩气缸伸出条件
AND T0111  ; RK_04 电芯除尘伸缩气缸伸出延时[A]
OR 600.11  ; RK_04 电芯除尘伸缩气缸伸出[A]
ANDLD
ANDNOT 500.10  ; RK_04 电芯除尘伸缩气缸缩回条件
ANDNOT 300.11  ; RK_04 电芯除尘伸缩气缸伸出[Pls]
ANDNOT 300.10  ; RK_04 电芯除尘伸缩气缸缩回[Pls]
ANDNOT 800.11  ; RK_04 电芯除尘伸缩气缸伸出位标志[0000.11]
LD H15.00  ; RK_02 U0_Y 电芯进料X轴回原点记忆
ANDNOT 851.02  ; RK_02 U0_Y 电芯进料X轴扫码OK放料位标志
ANDNOT 2011.13  ; RK_02 U0_Y 电芯进料X轴忙标志位
ANDNOT W206.15  ; RK_02 U0_Y 电芯进料X轴轴忙标志
LD H15.01  ; RK_02 U0_Z 电芯进料Z轴回原点记忆
AND 852.00  ; RK_02 U0_Z 电芯进料Z轴待料位（扫码）标志
ANDNOT 2014.13  ; RK_02 U0_Z 电芯进料Z轴忙标志位
ANDNOT W206.14  ; RK_02 U0_Z 电芯进料Z轴轴忙标志
ORLD
ANDLD
OUT 600.11  ; RK_04 电芯除尘伸缩气缸伸出[A]

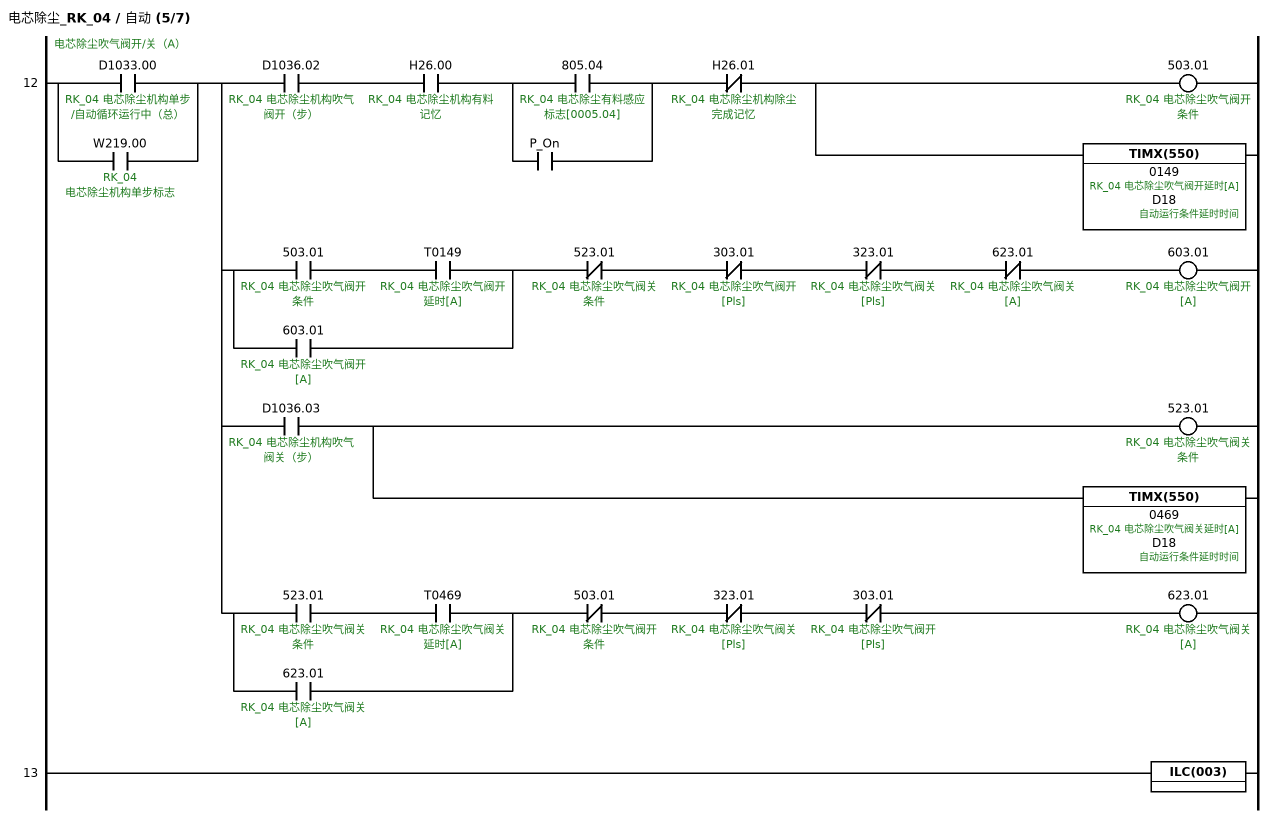
; rung 12: 电芯除尘吹气阀开/关（A）
LD D1033.00  ; RK_04 电芯除尘机构单步/自动循环运行中（总）
OR W219.00  ; RK_04  电芯除尘机构单步标志
OUT TR0
AND D1036.02  ; RK_04 电芯除尘机构吹气阀开（步）
AND H26.00  ; RK_04 电芯除尘机构有料记忆
LD 805.04  ; RK_04 电芯除尘有料感应标志[0005.04]
OR P_On
ANDLD
ANDNOT H26.01  ; RK_04 电芯除尘机构除尘完成记忆
OUT 503.01  ; RK_04 电芯除尘吹气阀开条件
TIMX(550) 0149 D18  ; 自动运行条件延时时间, RK_04 电芯除尘吹气阀开延时[A]
LD TR0
LD 503.01  ; RK_04 电芯除尘吹气阀开条件
AND T0149  ; RK_04 电芯除尘吹气阀开延时[A]
OR 603.01  ; RK_04 电芯除尘吹气阀开[A]
ANDLD
ANDNOT 523.01  ; RK_04 电芯除尘吹气阀关条件
ANDNOT 303.01  ; RK_04 电芯除尘吹气阀开[Pls]
ANDNOT 323.01  ; RK_04 电芯除尘吹气阀关[Pls]
ANDNOT 623.01  ; RK_04 电芯除尘吹气阀关[A]
OUT 603.01  ; RK_04 电芯除尘吹气阀开[A]
LD TR0
AND D1036.03  ; RK_04 电芯除尘机构吹气阀关（步）
OUT 523.01  ; RK_04 电芯除尘吹气阀关条件
TIMX(550) 0469 D18  ; 自动运行条件延时时间, RK_04 电芯除尘吹气阀关延时[A]
LD TR0
LD 523.01  ; RK_04 电芯除尘吹气阀关条件
AND T0469  ; RK_04 电芯除尘吹气阀关延时[A]
OR 623.01  ; RK_04 电芯除尘吹气阀关[A]
ANDLD
ANDNOT 503.01  ; RK_04 电芯除尘吹气阀开条件
ANDNOT 323.01  ; RK_04 电芯除尘吹气阀关[Pls]
ANDNOT 303.01  ; RK_04 电芯除尘吹气阀开[Pls]
OUT 623.01  ; RK_04 电芯除尘吹气阀关[A]
; rung 13
ILC(003)

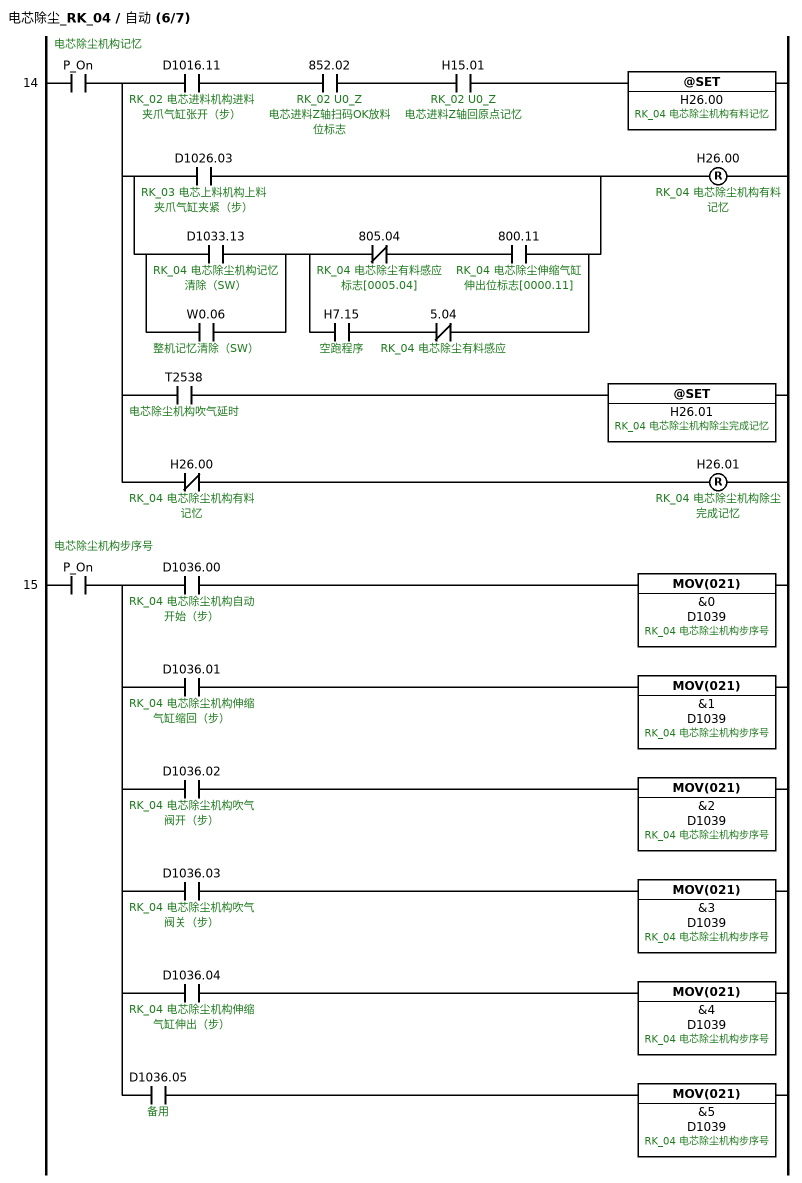
; rung 14: 电芯除尘机构记忆
LD P_On
OUT TR0
AND D1016.11  ; RK_02 电芯进料机构进料夹爪气缸张开（步）
AND 852.02  ; RK_02 U0_Z 电芯进料Z轴扫码OK放料位标志
AND H15.01  ; RK_02 U0_Z 电芯进料Z轴回原点记忆
@SET H26.00  ; RK_04 电芯除尘机构有料记忆
LD TR0
LD D1026.03  ; RK_03 电芯上料机构上料夹爪气缸夹紧（步）
LD D1033.13  ; RK_04 电芯除尘机构记忆清除（SW）
OR W0.06  ; 整机记忆清除（SW）
LDNOT 805.04  ; RK_04 电芯除尘有料感应标志[0005.04]
AND 800.11  ; RK_04 电芯除尘伸缩气缸伸出位标志[0000.11]
LD H7.15  ; 空跑程序
ANDNOT 5.04  ; RK_04 电芯除尘有料感应
ORLD
ANDLD
ORLD
ANDLD
RSET H26.00  ; RK_04 电芯除尘机构有料记忆
LD TR0
AND T2538  ; 电芯除尘机构吹气延时
@SET H26.01  ; RK_04 电芯除尘机构除尘完成记忆
LD TR0
ANDNOT H26.00  ; RK_04 电芯除尘机构有料记忆
RSET H26.01  ; RK_04 电芯除尘机构除尘完成记忆
; rung 15: 电芯除尘机构步序号
LD P_On
OUT TR0
AND D1036.00  ; RK_04 电芯除尘机构自动开始（步）
MOV(021) &0 D1039  ; RK_04 电芯除尘机构步序号
LD TR0
AND D1036.01  ; RK_04 电芯除尘机构伸缩气缸缩回（步）
MOV(021) &1 D1039  ; RK_04 电芯除尘机构步序号
LD TR0
AND D1036.02  ; RK_04 电芯除尘机构吹气阀开（步）
MOV(021) &2 D1039  ; RK_04 电芯除尘机构步序号
LD TR0
AND D1036.03  ; RK_04 电芯除尘机构吹气阀关（步）
MOV(021) &3 D1039  ; RK_04 电芯除尘机构步序号
LD TR0
AND D1036.04  ; RK_04 电芯除尘机构伸缩气缸伸出（步）
MOV(021) &4 D1039  ; RK_04 电芯除尘机构步序号
LD TR0
AND D1036.05  ; 备用
MOV(021) &5 D1039  ; RK_04 电芯除尘机构步序号

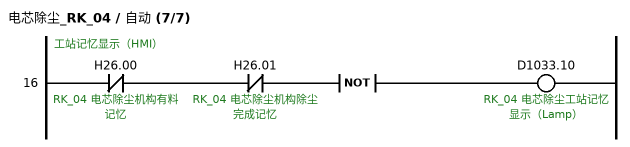
; rung 16: 工站记忆显示（HMI）
LDNOT H26.00  ; RK_04 电芯除尘机构有料记忆
ANDNOT H26.01  ; RK_04 电芯除尘机构除尘完成记忆
NOT(520)
OUT D1033.10  ; RK_04 电芯除尘工站记忆显示（Lamp）

### Section 复位

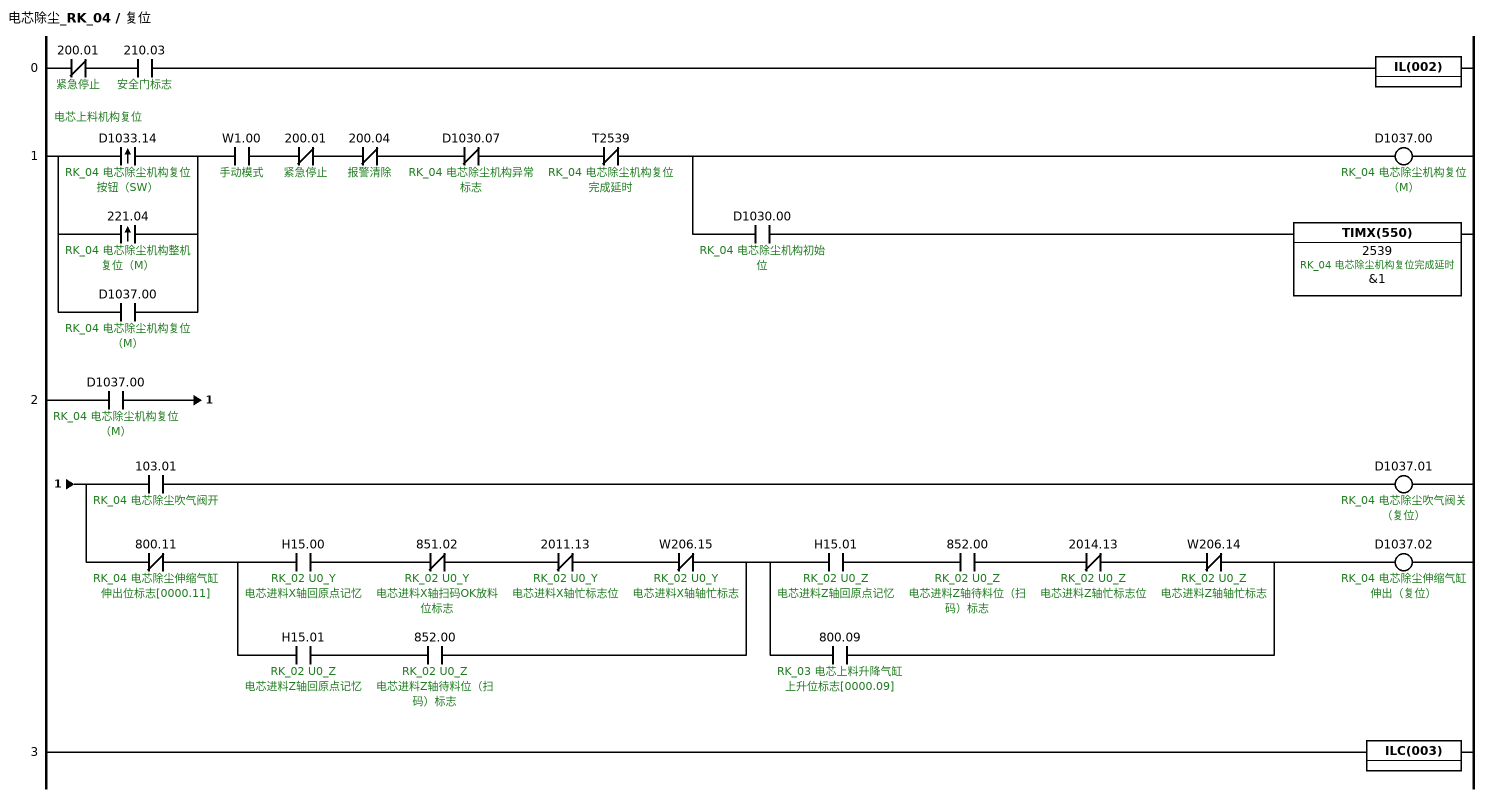
; rung 0
LDNOT 200.01  ; 紧急停止
AND 210.03  ; 安全门标志
IL(002)
; rung 1: 电芯上料机构复位
@LD D1033.14  ; RK_04 电芯除尘机构复位按钮（SW）
@OR 221.04  ; RK_04 电芯除尘机构整机复位（M）
OR D1037.00  ; RK_04 电芯除尘机构复位（M）
AND W1.00  ; 手动模式
ANDNOT 200.01  ; 紧急停止
ANDNOT 200.04  ; 报警清除
ANDNOT D1030.07  ; RK_04 电芯除尘机构异常标志
ANDNOT T2539  ; RK_04 电芯除尘机构复位完成延时
OUT D1037.00  ; RK_04 电芯除尘机构复位（M）
AND D1030.00  ; RK_04 电芯除尘机构初始位
TIMX(550) 2539 &1  ; RK_04 电芯除尘机构复位完成延时
; rung 2
LD D1037.00  ; RK_04 电芯除尘机构复位（M）
OUT TR0
AND 103.01  ; RK_04 电芯除尘吹气阀开
OUT D1037.01  ; RK_04 电芯除尘吹气阀关（复位）
LD TR0
ANDNOT 800.11  ; RK_04 电芯除尘伸缩气缸伸出位标志[0000.11]
LD H15.00  ; RK_02 U0_Y 电芯进料X轴回原点记忆
ANDNOT 851.02  ; RK_02 U0_Y 电芯进料X轴扫码OK放料位标志
ANDNOT 2011.13  ; RK_02 U0_Y 电芯进料X轴忙标志位
ANDNOT W206.15  ; RK_02 U0_Y 电芯进料X轴轴忙标志
LD H15.01  ; RK_02 U0_Z 电芯进料Z轴回原点记忆
AND 852.00  ; RK_02 U0_Z 电芯进料Z轴待料位（扫码）标志
ORLD
ANDLD
LD H15.01  ; RK_02 U0_Z 电芯进料Z轴回原点记忆
AND 852.00  ; RK_02 U0_Z 电芯进料Z轴待料位（扫码）标志
ANDNOT 2014.13  ; RK_02 U0_Z 电芯进料Z轴忙标志位
ANDNOT W206.14  ; RK_02 U0_Z 电芯进料Z轴轴忙标志
OR 800.09  ; RK_03 电芯上料升降气缸上升位标志[0000.09]
ANDLD
OUT D1037.02  ; RK_04 电芯除尘伸缩气缸伸出（复位）
; rung 3
ILC(003)

### Section 指示灯

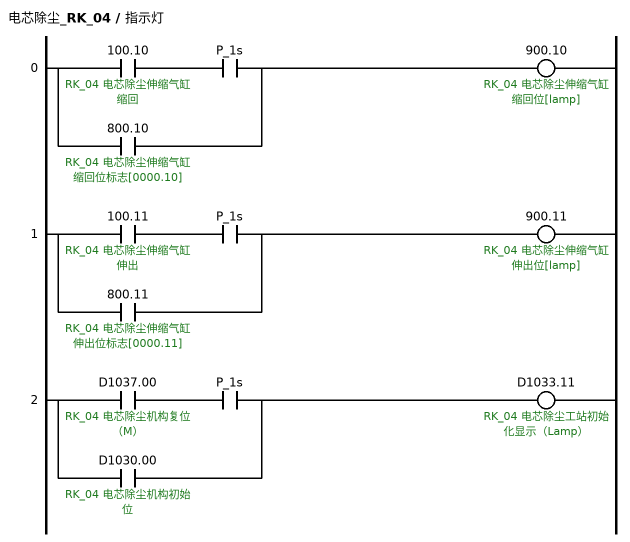
; rung 0
LD 100.10  ; RK_04 电芯除尘伸缩气缸缩回
AND P_1s
OR 800.10  ; RK_04 电芯除尘伸缩气缸缩回位标志[0000.10]
OUT 900.10  ; RK_04 电芯除尘伸缩气缸缩回位[lamp]
; rung 1
LD 100.11  ; RK_04 电芯除尘伸缩气缸伸出
AND P_1s
OR 800.11  ; RK_04 电芯除尘伸缩气缸伸出位标志[0000.11]
OUT 900.11  ; RK_04 电芯除尘伸缩气缸伸出位[lamp]
; rung 2
LD D1037.00  ; RK_04 电芯除尘机构复位（M）
AND P_1s
OR D1030.00  ; RK_04 电芯除尘机构初始位
OUT D1033.11  ; RK_04 电芯除尘工站初始化显示（Lamp）

### Section 外部输出

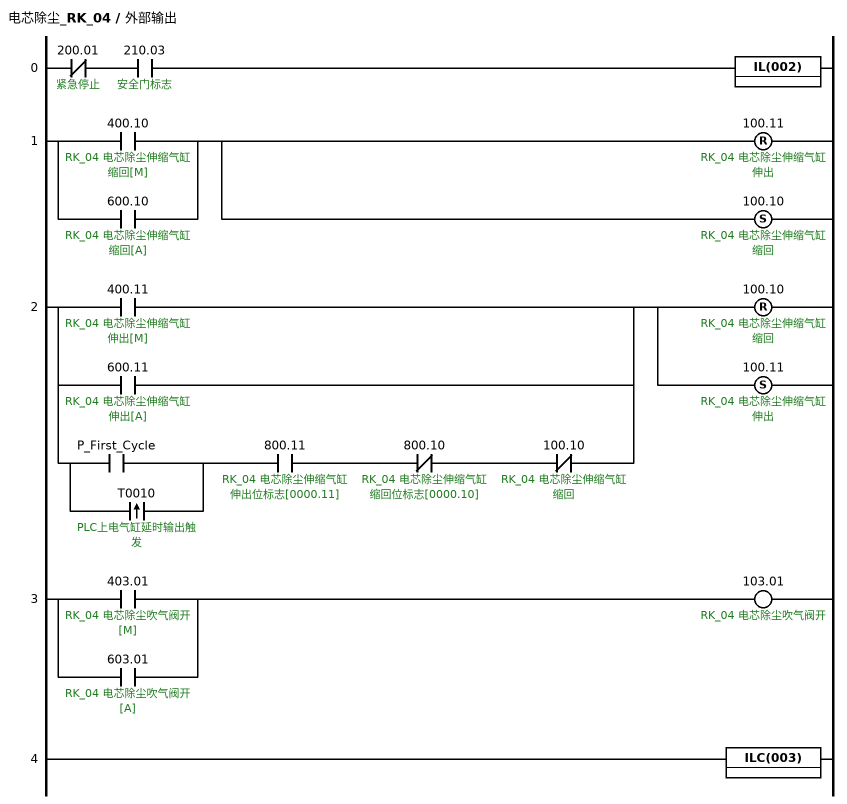
; rung 0
LDNOT 200.01  ; 紧急停止
AND 210.03  ; 安全门标志
IL(002)
; rung 1
LD 400.10  ; RK_04 电芯除尘伸缩气缸缩回[M]
OR 600.10  ; RK_04 电芯除尘伸缩气缸缩回[A]
RSET 100.11  ; RK_04 电芯除尘伸缩气缸伸出
SET 100.10  ; RK_04 电芯除尘伸缩气缸缩回
; rung 2
LD 400.11  ; RK_04 电芯除尘伸缩气缸伸出[M]
OR 600.11  ; RK_04 电芯除尘伸缩气缸伸出[A]
LD P_First_Cycle
@OR T0010  ; PLC上电气缸延时输出触发
AND 800.11  ; RK_04 电芯除尘伸缩气缸伸出位标志[0000.11]
ANDNOT 800.10  ; RK_04 电芯除尘伸缩气缸缩回位标志[0000.10]
ANDNOT 100.10  ; RK_04 电芯除尘伸缩气缸缩回
ORLD
RSET 100.10  ; RK_04 电芯除尘伸缩气缸缩回
SET 100.11  ; RK_04 电芯除尘伸缩气缸伸出
; rung 3
LD 403.01  ; RK_04 电芯除尘吹气阀开[M]
OR 603.01  ; RK_04 电芯除尘吹气阀开[A]
OUT 103.01  ; RK_04 电芯除尘吹气阀开
; rung 4
ILC(003)

### Section END
; rung 0
END(001)

## Program 入壳_RK_05 (cyclic task 5)

### Section Main_1入壳

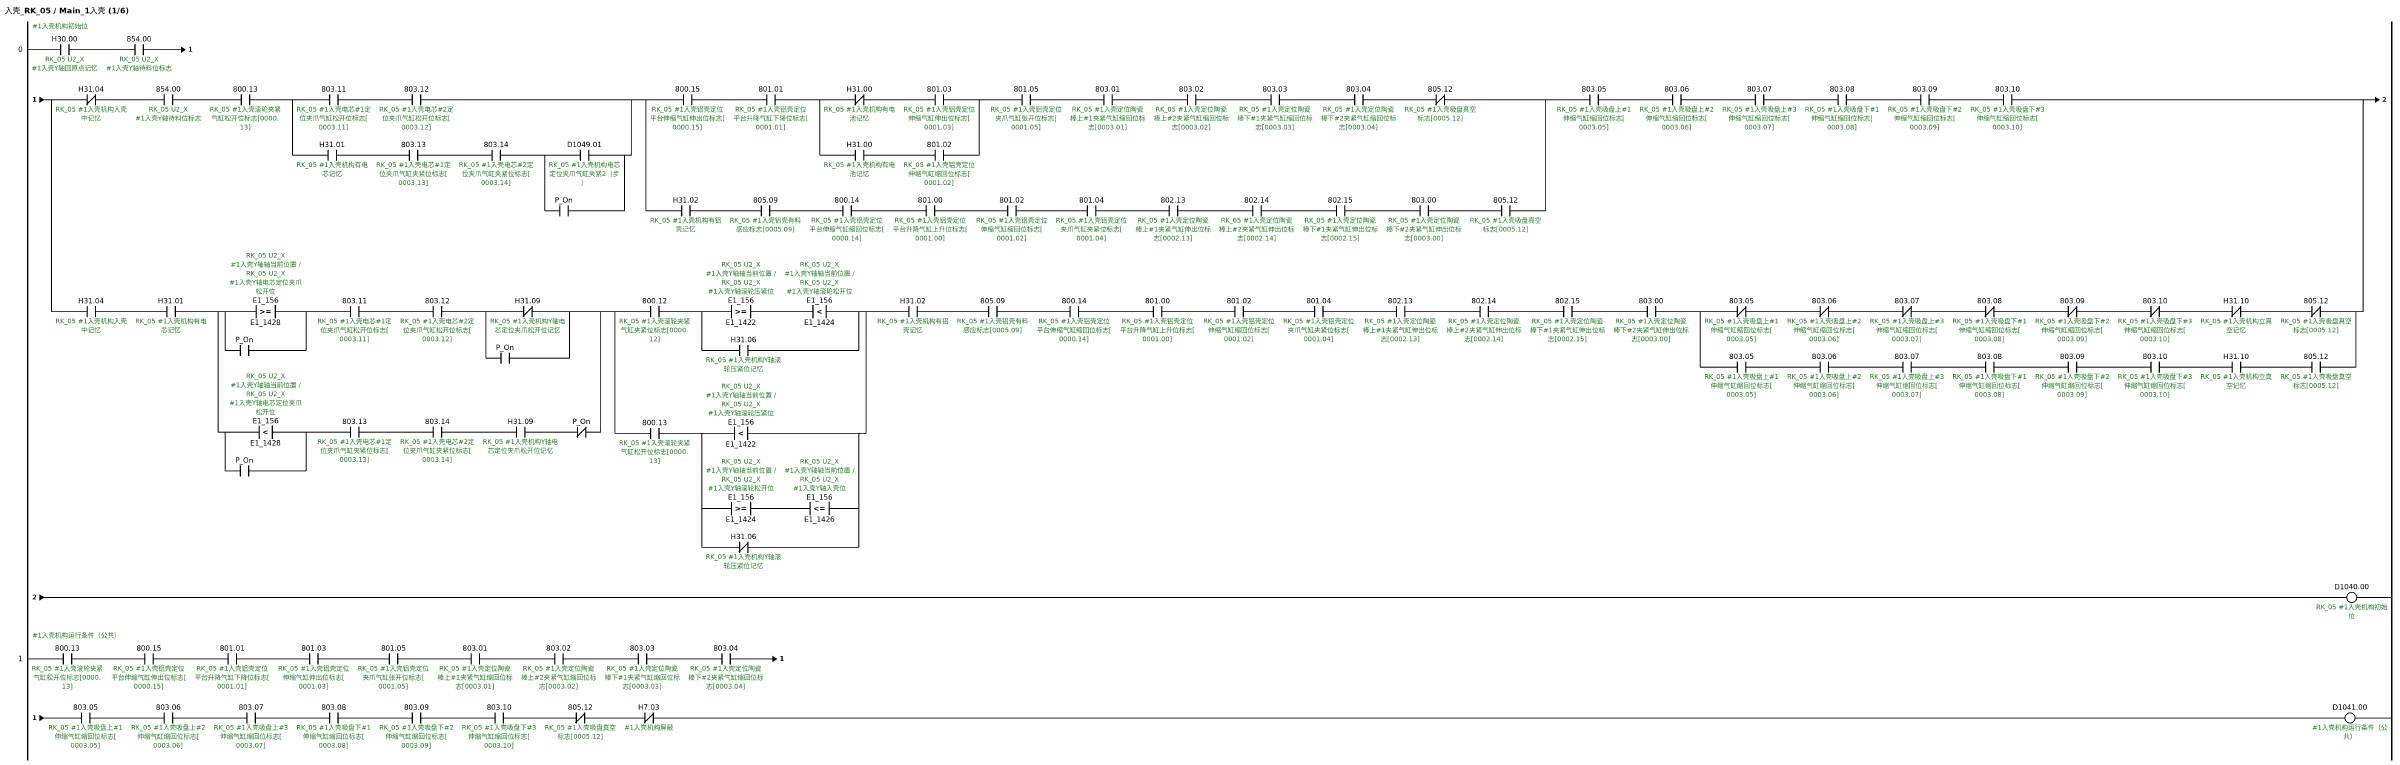
; rung 0: #1入壳机构初始位
LD H30.00  ; RK_05 U2_X #1入壳Y轴回原点记忆
AND 854.00  ; RK_05 U2_X #1入壳Y轴待料位标志
LDNOT H31.04  ; RK_05 #1入壳机构入壳中记忆
AND 854.00  ; RK_05 U2_X #1入壳Y轴待料位标志
AND 800.13  ; RK_05 #1入壳滚轮夹紧气缸松开位标志[0000.13]
LD 803.11  ; RK_05 #1入壳电芯#1定位夹爪气缸松开位标志[0003.11]
AND 803.12  ; RK_05 #1入壳电芯#2定位夹爪气缸松开位标志[0003.12]
LD H31.01  ; RK_05 #1入壳机构有电芯记忆
AND 803.13  ; RK_05 #1入壳电芯#1定位夹爪气缸夹紧位标志[0003.13]
AND 803.14  ; RK_05 #1入壳电芯#2定位夹爪气缸夹紧位标志[0003.14]
LD D1049.01  ; RK_05 #1入壳机构电芯定位夹爪气缸夹紧2（步）
OR P_On
ANDLD
ORLD
ANDLD
LD 800.15  ; RK_05 #1入壳铝壳定位平台伸缩气缸伸出位标志[0000.15]
AND 801.01  ; RK_05 #1入壳铝壳定位平台升降气缸下降位标志[0001.01]
LDNOT H31.00  ; RK_05 #1入壳机构有电池记忆
AND 801.03  ; RK_05 #1入壳铝壳定位伸缩气缸伸出位标志[0001.03]
LD H31.00  ; RK_05 #1入壳机构有电池记忆
AND 801.02  ; RK_05 #1入壳铝壳定位伸缩气缸缩回位标志[0001.02]
ORLD
ANDLD
AND 801.05  ; RK_05 #1入壳铝壳定位夹爪气缸张开位标志[0001.05]
AND 803.01  ; RK_05 #1入壳定位陶瓷棒上#1夹紧气缸缩回位标志[0003.01]
AND 803.02  ; RK_05 #1入壳定位陶瓷棒上#2夹紧气缸缩回位标志[0003.02]
AND 803.03  ; RK_05 #1入壳定位陶瓷棒下#1夹紧气缸缩回位标志[0003.03]
AND 803.04  ; RK_05 #1入壳定位陶瓷棒下#2夹紧气缸缩回位标志[0003.04]
ANDNOT 805.12  ; RK_05 #1入壳吸盘真空标志[0005.12]
LD H31.02  ; RK_05 #1入壳机构有铝壳记忆  // 20181014新增
AND 805.09  ; RK_05 #1入壳铝壳有料感应标志[0005.09]
AND 800.14  ; RK_05 #1入壳铝壳定位平台伸缩气缸缩回位标志[0000.14]
AND 801.00  ; RK_05 #1入壳铝壳定位平台升降气缸上升位标志[0001.00]
AND 801.02  ; RK_05 #1入壳铝壳定位伸缩气缸缩回位标志[0001.02]
AND 801.04  ; RK_05 #1入壳铝壳定位夹爪气缸夹紧位标志[0001.04]
AND 802.13  ; RK_05 #1入壳定位陶瓷棒上#1夹紧气缸伸出位标志[0002.13]
AND 802.14  ; RK_05 #1入壳定位陶瓷棒上#2夹紧气缸伸出位标志[0002.14]
AND 802.15  ; RK_05 #1入壳定位陶瓷棒下#1夹紧气缸伸出位标志[0002.15]
AND 803.00  ; RK_05 #1入壳定位陶瓷棒下#2夹紧气缸伸出位标志[0003.00]
AND 805.12  ; RK_05 #1入壳吸盘真空标志[0005.12]
ORLD
ANDLD
AND 803.05  ; RK_05 #1入壳吸盘上#1伸缩气缸缩回位标志[0003.05]
AND 803.06  ; RK_05 #1入壳吸盘上#2伸缩气缸缩回位标志[0003.06]
AND 803.07  ; RK_05 #1入壳吸盘上#3伸缩气缸缩回位标志[0003.07]
AND 803.08  ; RK_05 #1入壳吸盘下#1伸缩气缸缩回位标志[0003.08]
AND 803.09  ; RK_05 #1入壳吸盘下#2伸缩气缸缩回位标志[0003.09]
AND 803.10  ; RK_05 #1入壳吸盘下#3伸缩气缸缩回位标志[0003.10]
LD H31.04  ; RK_05 #1入壳机构入壳中记忆
AND H31.01  ; RK_05 #1入壳机构有电芯记忆
LD>=SL(328) E1_156 E1_1428  ; RK_05 U2_X #1入壳Y轴轴当前位置, RK_05 U2_X #1入壳Y轴电芯定位夹爪松开位
OR P_On
AND 803.11  ; RK_05 #1入壳电芯#1定位夹爪气缸松开位标志[0003.11]
AND 803.12  ; RK_05 #1入壳电芯#2定位夹爪气缸松开位标志[0003.12]
LDNOT H31.09  ; RK_05 #1入壳机构Y轴电芯定位夹爪松开位记忆
OR P_On
ANDLD
LD<SL(313) E1_156 E1_1428  ; RK_05 U2_X #1入壳Y轴轴当前位置, RK_05 U2_X #1入壳Y轴电芯定位夹爪松开位
OR P_On
AND 803.13  ; RK_05 #1入壳电芯#1定位夹爪气缸夹紧位标志[0003.13]
AND 803.14  ; RK_05 #1入壳电芯#2定位夹爪气缸夹紧位标志[0003.14]
AND H31.09  ; RK_05 #1入壳机构Y轴电芯定位夹爪松开位记忆
ANDNOT P_On
ORLD
ANDLD
LD 800.12  ; RK_05 #1入壳滚轮夹紧气缸夹紧位标志[0000.12]
LD>=SL(328) E1_156 E1_1422  ; RK_05 U2_X #1入壳Y轴轴当前位置, RK_05 U2_X #1入壳Y轴滚轮压紧位
AND<SL(313) E1_156 E1_1424  ; RK_05 U2_X #1入壳Y轴轴当前位置, RK_05 U2_X #1入壳Y轴滚轮松开位
OR H31.06  ; RK_05 #1入壳机构Y轴滚轮压紧位记忆
ANDLD
LD 800.13  ; RK_05 #1入壳滚轮夹紧气缸松开位标志[0000.13]
LD<SL(313) E1_156 E1_1422  ; RK_05 U2_X #1入壳Y轴轴当前位置, RK_05 U2_X #1入壳Y轴滚轮压紧位
LD>=SL(328) E1_156 E1_1424  ; RK_05 U2_X #1入壳Y轴轴当前位置, RK_05 U2_X #1入壳Y轴滚轮松开位
AND<=SL(318) E1_156 E1_1426  ; RK_05 U2_X #1入壳Y轴轴当前位置, RK_05 U2_X #1入壳Y轴入壳位
ORLD
ORNOT H31.06  ; RK_05 #1入壳机构Y轴滚轮压紧位记忆
ANDLD
ORLD
ANDLD
AND H31.02  ; RK_05 #1入壳机构有铝壳记忆
AND 805.09  ; RK_05 #1入壳铝壳有料感应标志[0005.09]
AND 800.14  ; RK_05 #1入壳铝壳定位平台伸缩气缸缩回位标志[0000.14]
AND 801.00  ; RK_05 #1入壳铝壳定位平台升降气缸上升位标志[0001.00]
AND 801.02  ; RK_05 #1入壳铝壳定位伸缩气缸缩回位标志[0001.02]
AND 801.04  ; RK_05 #1入壳铝壳定位夹爪气缸夹紧位标志[0001.04]
AND 802.13  ; RK_05 #1入壳定位陶瓷棒上#1夹紧气缸伸出位标志[0002.13]
AND 802.14  ; RK_05 #1入壳定位陶瓷棒上#2夹紧气缸伸出位标志[0002.14]
AND 802.15  ; RK_05 #1入壳定位陶瓷棒下#1夹紧气缸伸出位标志[0002.15]
AND 803.00  ; RK_05 #1入壳定位陶瓷棒下#2夹紧气缸伸出位标志[0003.00]
LDNOT 803.05  ; RK_05 #1入壳吸盘上#1伸缩气缸缩回位标志[0003.05]
ANDNOT 803.06  ; RK_05 #1入壳吸盘上#2伸缩气缸缩回位标志[0003.06]
ANDNOT 803.07  ; RK_05 #1入壳吸盘上#3伸缩气缸缩回位标志[0003.07]
ANDNOT 803.08  ; RK_05 #1入壳吸盘下#1伸缩气缸缩回位标志[0003.08]
ANDNOT 803.09  ; RK_05 #1入壳吸盘下#2伸缩气缸缩回位标志[0003.09]
ANDNOT 803.10  ; RK_05 #1入壳吸盘下#3伸缩气缸缩回位标志[0003.10]
ANDNOT H31.10  ; RK_05 #1入壳机构立真空记忆
ANDNOT 805.12  ; RK_05 #1入壳吸盘真空标志[0005.12]
LD 803.05  ; RK_05 #1入壳吸盘上#1伸缩气缸缩回位标志[0003.05]
AND 803.06  ; RK_05 #1入壳吸盘上#2伸缩气缸缩回位标志[0003.06]
AND 803.07  ; RK_05 #1入壳吸盘上#3伸缩气缸缩回位标志[0003.07]
AND 803.08  ; RK_05 #1入壳吸盘下#1伸缩气缸缩回位标志[0003.08]
AND 803.09  ; RK_05 #1入壳吸盘下#2伸缩气缸缩回位标志[0003.09]
AND 803.10  ; RK_05 #1入壳吸盘下#3伸缩气缸缩回位标志[0003.10]
AND H31.10  ; RK_05 #1入壳机构立真空记忆
AND 805.12  ; RK_05 #1入壳吸盘真空标志[0005.12]
ORLD
ANDLD
ORLD
ANDLD
OUT D1040.00  ; RK_05 #1入壳机构初始位
; rung 1: #1入壳机构运行条件（公共）
LD 800.13  ; RK_05 #1入壳滚轮夹紧气缸松开位标志[0000.13]
AND 800.15  ; RK_05 #1入壳铝壳定位平台伸缩气缸伸出位标志[0000.15]
AND 801.01  ; RK_05 #1入壳铝壳定位平台升降气缸下降位标志[0001.01]
AND 801.03  ; RK_05 #1入壳铝壳定位伸缩气缸伸出位标志[0001.03]
AND 801.05  ; RK_05 #1入壳铝壳定位夹爪气缸张开位标志[0001.05]
AND 803.01  ; RK_05 #1入壳定位陶瓷棒上#1夹紧气缸缩回位标志[0003.01]
AND 803.02  ; RK_05 #1入壳定位陶瓷棒上#2夹紧气缸缩回位标志[0003.02]
AND 803.03  ; RK_05 #1入壳定位陶瓷棒下#1夹紧气缸缩回位标志[0003.03]
AND 803.04  ; RK_05 #1入壳定位陶瓷棒下#2夹紧气缸缩回位标志[0003.04]
AND 803.05  ; RK_05 #1入壳吸盘上#1伸缩气缸缩回位标志[0003.05]
AND 803.06  ; RK_05 #1入壳吸盘上#2伸缩气缸缩回位标志[0003.06]
AND 803.07  ; RK_05 #1入壳吸盘上#3伸缩气缸缩回位标志[0003.07]
AND 803.08  ; RK_05 #1入壳吸盘下#1伸缩气缸缩回位标志[0003.08]
AND 803.09  ; RK_05 #1入壳吸盘下#2伸缩气缸缩回位标志[0003.09]
AND 803.10  ; RK_05 #1入壳吸盘下#3伸缩气缸缩回位标志[0003.10]
ANDNOT 805.12  ; RK_05 #1入壳吸盘真空标志[0005.12]
ANDNOT H7.03  ; #1入壳机构屏蔽
OUT D1041.00  ; #1入壳机构运行条件（公共）

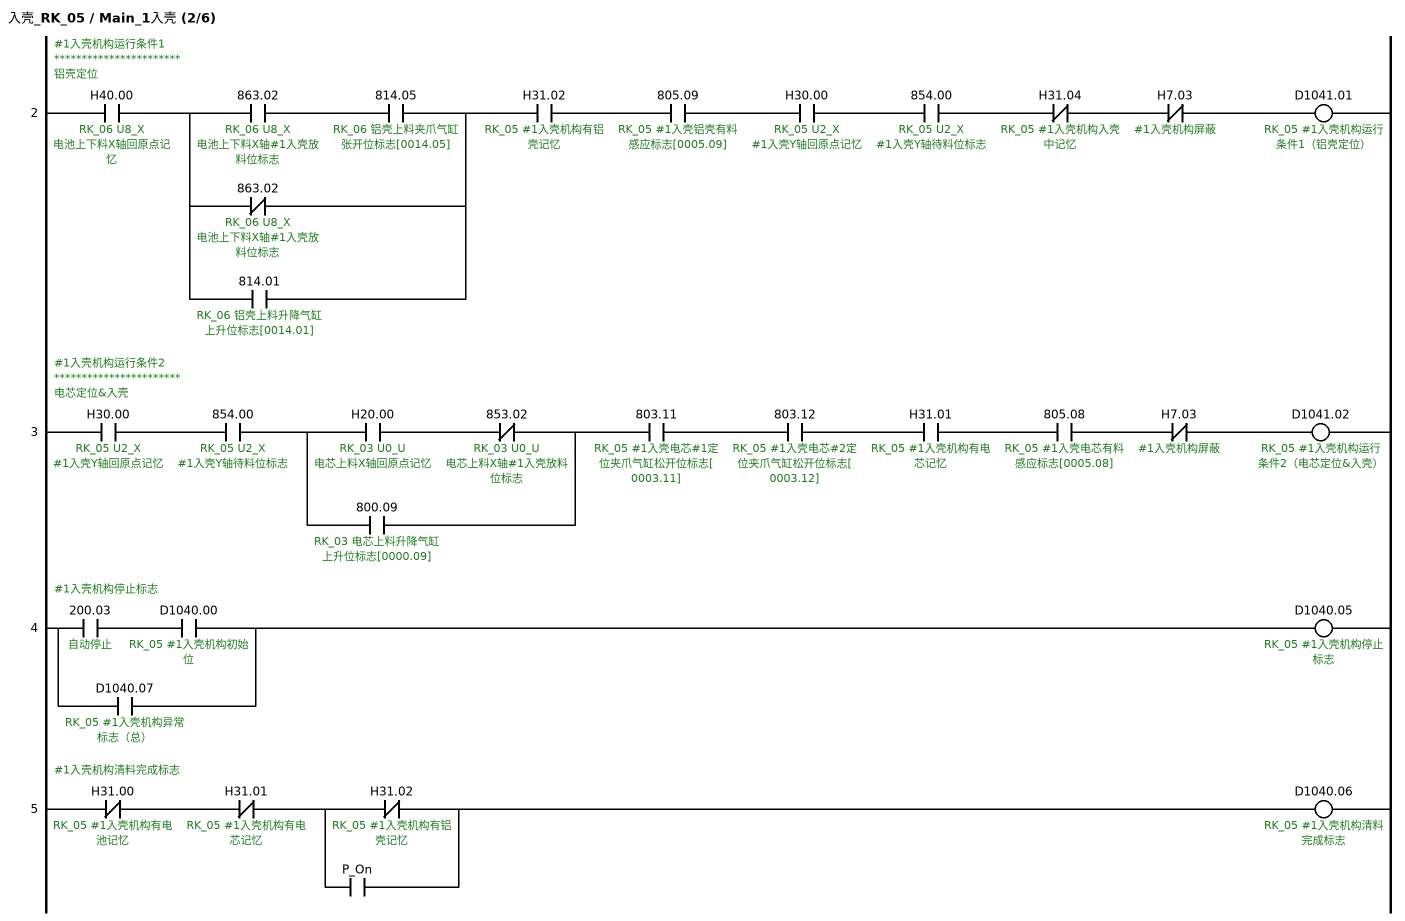
; rung 2: #1入壳机构运行条件1 / *********************** / 铝壳定位
LD H40.00  ; RK_06 U8_X 电池上下料X轴回原点记忆
LD 863.02  ; RK_06 U8_X 电池上下料X轴#1入壳放料位标志
AND 814.05  ; RK_06 铝壳上料夹爪气缸张开位标志[0014.05]
ORNOT 863.02  ; RK_06 U8_X 电池上下料X轴#1入壳放料位标志
OR 814.01  ; RK_06 铝壳上料升降气缸上升位标志[0014.01]
ANDLD
AND H31.02  ; RK_05 #1入壳机构有铝壳记忆
AND 805.09  ; RK_05 #1入壳铝壳有料感应标志[0005.09]
AND H30.00  ; RK_05 U2_X #1入壳Y轴回原点记忆
AND 854.00  ; RK_05 U2_X #1入壳Y轴待料位标志
ANDNOT H31.04  ; RK_05 #1入壳机构入壳中记忆
ANDNOT H7.03  ; #1入壳机构屏蔽
OUT D1041.01  ; RK_05 #1入壳机构运行条件1（铝壳定位）
; rung 3: #1入壳机构运行条件2 / *********************** / 电芯定位&入壳
LD H30.00  ; RK_05 U2_X #1入壳Y轴回原点记忆
AND 854.00  ; RK_05 U2_X #1入壳Y轴待料位标志
LD H20.00  ; RK_03 U0_U 电芯上料X轴回原点记忆
ANDNOT 853.02  ; RK_03 U0_U 电芯上料X轴#1入壳放料位标志
OR 800.09  ; RK_03 电芯上料升降气缸上升位标志[0000.09]
ANDLD
AND 803.11  ; RK_05 #1入壳电芯#1定位夹爪气缸松开位标志[0003.11]
AND 803.12  ; RK_05 #1入壳电芯#2定位夹爪气缸松开位标志[0003.12]
AND H31.01  ; RK_05 #1入壳机构有电芯记忆
AND 805.08  ; RK_05 #1入壳电芯有料感应标志[0005.08]
ANDNOT H7.03  ; #1入壳机构屏蔽
OUT D1041.02  ; RK_05 #1入壳机构运行条件2（电芯定位&入壳）
; rung 4: #1入壳机构停止标志
LD 200.03  ; 自动停止
AND D1040.00  ; RK_05 #1入壳机构初始位
OR D1040.07  ; RK_05 #1入壳机构异常标志（总）
OUT D1040.05  ; RK_05 #1入壳机构停止标志
; rung 5: #1入壳机构清料完成标志
LDNOT H31.00  ; RK_05 #1入壳机构有电池记忆
ANDNOT H31.01  ; RK_05 #1入壳机构有电芯记忆
LDNOT H31.02  ; RK_05 #1入壳机构有铝壳记忆
OR P_On
ANDLD
OUT D1040.06  ; RK_05 #1入壳机构清料完成标志

